(*
Nazwa:			VIS
Opis:			Zmienne wykorzystywane i zmieniane tylko z wizualizacji
Wersja:			v0.2
Data:			2024-02-06
Autor:			DP,MP
Urzadzenia:		
Konfiguracja:	
Info:
Zmiany:
- 20240205 [DP] Poprawki przed nowa wizką
*)

{attribute 'qualified_only'}

VAR_GLOBAL	
	
(********DANE MASZYNY***********)
sType: STRING[255];
sSerialNumber: STRING[255];
rProgramVersion: REAL;
rLastTimeChanges: REAL;
(*******************************)	

    (* OPISY ZMIENNYCH TYPU INT DO POŚWWIETLANIA STANÓW STACJI
	E_PackMLState : 
					eUndefined				:=  0, //----Nieużywany
					eClearing 				:=  1, //----Nieużywany
					eStopped 				:=  2, //Błąd
					eStarting 				:=  3, //Uruchamianie
					eIdle 					:=  4, //Postój
					eSuspended 				:=  5, //---Nieużywany
					eExecute 				:=  6, //Praca
					eStopping	 			:=  7, //Zatrzymywanie
					eAborting 				:=  8, //Zatrzymywanie awaryjne
					eAborted 				:=  9, //Zatrzymano awaryjnie
					eHolding 				:= 10, //---Nieużywany
					eHeld 					:= 11, //---Nieużywany
					eUnholding 				:= 12, //---Nieużywany
					eSuspending 			:= 13, //---Nieużywany
					eUnsuspending 			:= 14, //---Nieużywany
					eResetting 				:= 15, //Resetowanie błędu, bazowanie
					eCompleting 			:= 16, //---Nieużywany
					eComplete	 			:= 17  //---Nieużywany
	
	E_Station :
					eDisabled 				:= 0, // Stan nieaktywnosci (Stacja wyłączona)             
					eAborted 				:= 1, // Stan bezpiecznego zatrzymania (po Abortingu) 
					eAborting 				:= 2, // Stan bezpiecznego zatrzymywania (po EStopie)
					eError 					:= 3, // Stan błędu 		
					eResetting 				:= 4, // Stan resetowania bledu (po Errorze)		                
					eManualMovement 		:= 5, // Stan ruchów manualnych         
					eHoming 				:= 6, // Stan bazowania 
					eHomingDone 			:= 7, // Stan wykonania bazowania 
					ePreparingToReady 		:= 8, // Stan przygotowywania do gotowosci (zawsze przed Ready)           
					ePreparingToDisable 	:= 9, // Stan przygotowywania do nieaktywnosci (po wyłączeniu Enable)                               
					eReady					:= 10,// Stan gotowosci 
					eStopping 				:= 11,// Stan zatrzymywania 
					eStarting 				:= 12,// Stan uruchamiania (po Ready)
					eRunning 				:= 13 // Stan wykonywania cyklu (po Startingu), w tym stanie osobny 
					
					
	Legenda dla wizki :
	[H] - Hidden, prawdopodobnie nie potrzebne
	[I] - Info, informacja,
	[L] - Later, do zrobienia później, być może do przerobienia
	Uprawienia:
	brak opisu - operator
	[m] - Meechanik i powyżej
	[t] - Technolog i powyżej
	[s] - Serwis i powyżek
	[a] - Admin			
	*)
	(*****Zmienne ogólne****)
	
	(* Wykresy dozowania*)
	aPoints												: ARRAY [0..11,0..599] OF ST_Point;	// Sam wykres wybrando doziwniki + jego simulacji
	udiDossagerNum										: UDINT	:=	0;						// Wybrany dozownik 0 - pierwszy, 3 - czwarty
	bDrawChart											: BOOL;								// Cykl simulacji
	nDrawLenght										:INT;
	nTimeMarkerDSPh1                                :INT;
	nTimeMarkerDSPh2                                :INT;
	nTimeMarkerDSPh3                                :INT;
	nTimeMarkerDSPh4								:INT;
	nTimeMarkerDSPh5								:INT;
	aHorizontalChart								: ARRAY[0..4] OF ARRAY [0..0] OF INT;
	lrTorqMin										:LREAL;
	lrTorqMax										:LREAL;
	aWeightPoints									: ARRAY [0..7,0..9999] OF ST_Point_1;
	
	
	
	
	
	
	
	
	//Zmienne przejść do różnych stanów	
	iMachineState										:UINT;						// Stan maszyny
	sMachineState										:STRING; 					// Stan maszyny
	wsMachineState										:WSTRING; 					// Stan maszyny

	//Okno przezbrajania po wyborze receptury
	bMachinePartsChangeOver								:BOOL;						// Włączone przezbrajanie (ustawić z wizki)
	iMachinePartsChangeOver								:INT;						// Stan przezbrajania (0-ruch,1-pozycja gorna,-1-pozycja dolna) 
	bBottleSorterDisable								:BOOL:=FALSE;				// Wyłączenie sortera butelek
	bCapSorterDisable									:BOOL:=FALSE;				// Wyłączenie sortera nasadek
	
	//Ekran z komunikatami
	bDialogBoxOn										:BOOL;		 				// Wyświetl okno komunikatów
	bDialogBoxText										:STRING[255];				// Treść na oknie komunikatów 
	bDialogBoxText2										:STRING[255];				// Treść na oknie komunikatów (nie tłumaczone, zmienne)
	sDialogBoxPicture									:STRING[255];				// Nazwa obrazka który ma sie wyświetlać, '' - brak obrazu, 1,2,ok,info,uwaga 
																					// (odnosi się do pliku pictures.txt gdzie są podaje lokalizacje obrazków)
																					(*	[{"ImagePath":"c:\\img\\img1.png","ImageID":"1"}, 
																						{"ImagePath":"c:\\img\\img2.png","ImageID":"2"},
																						{"ImagePath":"c:\\img\\ok.png","ImageID":"ok"},
																						{"ImagePath":"c:\\img\\info.png","ImageID":"info"},
																						{"ImagePath":"c:\\img\\uwaga.png","ImageID":"uwaga"}] *)
	bDialogBoxAck										:BOOL;						// Przycisk OK
	bDialogBoxCancelAck									:BOOL;						// Przycisk ANULUJ
	nDialogBoxType										:UINT;						// Rodzaj okna, 0-nic, 1-tylko przycisk OK, 2 - tylko przycisk Anuluj, 3 - Przycisk OK i Anuluj
	bDialogBoxAckNeeded									:BOOL;						// [H] Potrzebne potwierdzenie					

	wsDialogBoxText										:WSTRING;				// Treść na oknie komunikatów 
	wsDialogBoxText2									:WSTRING;				// Treść na oknie komunikatów (nie tłumaczone, zmienne)
	
	//Wyświetlanie informacji na ekranie głównym
	//Przyczyny odrzuceń (wyświetlić na ekranie głównym bez dodatkowego odpisu)
	sBadPackageReason1									:STRING;					// Powód odrzutu butelek 		//sBadPackageReason1 sBadPackageReason1
	sBadPackageReason2									:STRING;					//								//sBadPackageReason2 sBadPackageReason2
	sBadPackageReason3									:STRING;					//								//sBadPackageReason3 sBadPackageReason3	
	iBadPackageReasonCount1								:INT;						// Ilość odrzuconych opakowań
	iBadPackageReasonCount2								:INT;						//
	iBadPackageReasonCount3								:INT;						//
	wsBadPackageReason1									:WSTRING;					// Powód odrzutu butelek 		//sBadPackageReason1 sBadPackageReason1
	wsBadPackageReason2									:WSTRING;					//								//sBadPackageReason2 sBadPackageReason2
	wsBadPackageReason3									:WSTRING;					//								//sBadPackageReason3 sBadPackageReason3	
	AStBadPackageReason									:ARRAY[0..63] OF S_Information;	// ID informacji do powodów odrzuceń
	bBadPackageReasonReset								:BOOL;						// Czyszczenie tablicy odrzuceń
	
	iNumbersOfFormsBetweenWeightAndScrewers				:INT;						// Ilość formatek pomiędzy wagą a zakręcarkami: zmienna
	
	sSlowestStation1									:STRING;					//	Najwolniejsza stacja nr 1	//sSlowestStation1 iSlowestStationCount1
	sSlowestStation2									:STRING;					//	Najwolniejsza stacja nr 2	//sSlowestStation2 iSlowestStationCount2
	sSlowestStation3									:STRING;					//	Najwolniejsza stacja nr 3	//itd.
	sSlowestStation4									:STRING;					//	Najwolniejsza stacja nr 4
	sSlowestStation5									:STRING;					//	Najwolniejsza stacja nr 5	
	iSlowestStationCount1								:INT;					  	//	Czas cyklu dla najwolniejszej stacji nr 1
	iSlowestStationCount2								:INT;					  	//	Czas cyklu dla najwolniejszej stacji nr 2
	iSlowestStationCount3								:INT;					  	//	Czas cyklu dla najwolniejszej stacji nr 3
	iSlowestStationCount4								:INT;					  	//	Czas cyklu dla najwolniejszej stacji nr 4
	iSlowestStationCount5								:INT;					  	//	Czas cyklu dla najwolniejszej stacji nr 5
	wsSlowestStation1									:WSTRING;					//	Najwolniejsza stacja nr 1	//sSlowestStation1 iSlowestStationCount1
	wsSlowestStation2									:WSTRING;					//	Najwolniejsza stacja nr 2	//sSlowestStation2 iSlowestStationCount2	
	wsSlowestStation3									:WSTRING;					//	Najwolniejsza stacja nr 3	//itd.	
	wsSlowestStation4									:WSTRING;					//	Najwolniejsza stacja nr 4	
	wsSlowestStation5									:WSTRING;					//	Najwolniejsza stacja nr 5	
	
	//Przyciski główne na HMI (wysuwany pasek lub na ekranie głównym)
	bDoorsUnlock										:BOOL;						// Otwórz drzwi 	
	bCycleReset											:BOOL;						// Reset cyklu 
	bCounterReset										:BOOL;						// Reset Liczników
	bConfectionEnding									:BOOL; 						// Zakończenie konfekcji
	bWeighingForm										:BOOL;						// [m] Przeważanie formatek
	bCapSorterEmptyingMode								:BOOL;						// Opróżnianie sortera nakrętek
	bBottleSorterEmptyingMode							:BOOL;						// Opróżnianie sortera butelek
	bBottleDeleteUnderDispencers						:BOOL;						// Usuń butelki pod dozownikami
	bSingleRealeseIfNoCapFromScrewers					:BOOL:=FALSE;						// Wypuszczanie pojedyńczo z zakręcarek jeżeli nie ma nasadki
	
	//Zmienne wystawiane z HMI
	bServiceMode										:BOOL; 						// Tryb serwisowy 
	bSimulation											:BOOL;						// [s] Przycisk trybu symulacyjnego
	bCheckStart 										:BOOL;						// Próba uruchomienia (PLC ustawia na 1, HMI na 0)
	bAllowStart 										:BOOL;						// Uruchomienie maszyny możliwe (HMI ustawia na 1 po bCheckStart i ktoś jest zalogowany, PLC ustawia na 0)
	iHMICommunication									:INT;						// [I] Licznik komunikacji, gdy się nie zmienia przez jakiś czas, wizka może wystawiać błąd
	bRecipeCalculate									:BOOL;						// Oblicz parametry receptury

	//[s] Zmienne tylko dla serwisu
	bWritePersistent									:BOOL; 						// [H] Zmienna zapisujaca wartosci zmiennych persistent
	bCycleStart											:BOOL;	(**)				// [H] Zdalny start/stop maszyny
	
	//Liczniki 
	uiCounterMachineEfficiency							:UINT; 						// Wydajność chwilowa maszyny[szt./h]
	uiCounterInstantEfficiency							:UINT; 						// Wydajność chwilowa prawidłowych butelek [szt./h]
	uiCounterAverageEfficiency							:UINT;						// Średnia wydajność [szt./h]
	udiCounterShiftBottles								:UDINT;						// Zmianowa ilość butelek [szt.]					
	uiCounterGoodBottles								:UINT;						// Prawidłowo napełnione opakowania [szt.]
	uiCounterBadBottles									:UINT;						// Odrzucone opakowania [szt]
	//Liczniki OEE
	udiCounterExecuteTime								:UINT;						// Cza pracy [min]
	udiCounterReadyTime									:UINT;						// Cza postoju [min]
	udiCounterErrorTime									:UINT;						// Cza błędu [min]
	
	//Lampki w trybie serwisowym pomocne do ustawiania stacji
	bCapPuttedCheckSensor								:BOOL;						// Czujnik nasadki przed zakręcarką
	bCapCorrectCheckCapOnSensor							:BOOL;						// Czujnik nasadki za zakręcarką
	bCapCorrectCheckCapNotScrewedSensor					:BOOL;						// Czujnik źle zakręconej nasadki

	(*Wykresy, statystyki, informacje*) 
	//Pomiary wag i dozowań do wyświetlenia na ekranie głównym
	lrDispencer1DoseVolumeCV							:LREAL;						// Doza 1 [ml]
	lrDispencer2DoseVolumeCV							:LREAL;						// Doza 2 [ml]
	lrDispencer3DoseVolumeCV							:LREAL;						// Doza 3 [ml]	
	lrDispencer4DoseVolumeCV							:LREAL;						// Doza 4 [ml]	
	lrDispencer1WeightMeasured							:LREAL;						// Waga z dozownika 1 [g]	
	lrDispencer2WeightMeasured							:LREAL;						// Waga z dozownika 2 [g]		
	lrDispencer3WeightMeasured							:LREAL;						// Waga z dozownika 3 [g]	
	lrDispencer4WeightMeasured							:LREAL;						// Waga z dozownika 4 [g]	
	bDispencer1WeightMeasured							:BOOL;						// [H] Waga zmierzona z dozownika nr 1	
	bDispencer2WeightMeasured							:BOOL;						// [H] Waga zmierzona z dozownika nr 2
	bDispencer3WeightMeasured							:BOOL;						// [H] Waga zmierzona z dozownika nr 3
	bDispencer4WeightMeasured							:BOOL;						// [H] Waga zmierzona z dozownika nr 4
		
	AsChartDose1										:ARRAY [0..500] OF STRING;	// [L] Wykres ostatniego dozowania 1 "Czas;PozycjaTłoka;PozycjaPodnośnika;ZawórSsący;ZaworDozujacy;Tacka" 
	AsChartDose2										:ARRAY [0..500] OF STRING;	// [L] Wykres ostatniego dozowania 2 "Czas;PozycjaTłoka;PozycjaPodnośnika;ZawórSsący;ZaworDozujacy;Tacka" 									
	AsChartDose3										:ARRAY [0..500] OF STRING;	// [L] Wykres ostatniego dozowania 3 "Czas;PozycjaTłoka;PozycjaPodnośnika;ZawórSsący;ZaworDozujacy;Tacka" 									
	AsChartDose4										:ARRAY [0..500] OF STRING;	// [L] Wykres ostatniego dozowania 4 "Czas;PozycjaTłoka;PozycjaPodnośnika;ZawórSsący;ZaworDozujacy;Tacka" 			
	AStAsChartDose1										:ARRAY [0..100] OF ARRAY [0..5,0..500] OF INT; // [L] Wykres ostatniego dozowania 1 "Czas;PozycjaTłoka;PozycjaPodnośnika;ZawórSsący;ZaworDozujacy;Tacka"
	AStAsChartDose2										:ARRAY [0..100] OF ARRAY [0..5,0..500] OF INT; // [L] Wykres ostatniego dozowania 1 "Czas;PozycjaTłoka;PozycjaPodnośnika;ZawórSsący;ZaworDozujacy;Tacka"
	AStAsChartDose3										:ARRAY [0..100] OF ARRAY [0..5,0..500] OF INT; // [L] Wykres ostatniego dozowania 1 "Czas;PozycjaTłoka;PozycjaPodnośnika;ZawórSsący;ZaworDozujacy;Tacka"
	AStAsChartDose4										:ARRAY [0..100] OF ARRAY [0..5,0..500] OF INT; // [L] Wykres ostatniego dozowania 1 "Czas;PozycjaTłoka;PozycjaPodnośnika;ZawórSsący;ZaworDozujacy;Tacka"
	
	
	AsChartGripperScrewer1								:ARRAY [0..500] OF STRING;	// [L] Wykres ostatniego zakręcania 1 "Czas;Wysokość;Obrót;Moment;SiłownikChwytania;;" 
	AsChartGripperScrewer2								:ARRAY [0..500] OF STRING;	// [L] Wykres ostatniego zakręcania 2 "Czas;Wysokość;Obrót;Moment;SiłownikChwytania;;" 
	AStChartGripperScrewer1								:ARRAY [0..100] OF ARRAY [0..5,0..500] OF INT;	// [L] Wykres ostatniego zakręcania 1 "Wysokość;Obrót;Prędkość;SiłownikChwytania;Czas;Pusty;;" 	
	AStChartGripperScrewer2								:ARRAY [0..100] OF ARRAY [0..5,0..500] OF INT;	// [L] Wykres ostatniego zakręcania 2 "Wysokość;Obrót;Prędkość;SiłownikChwytania;Czas;Pusty;;" 
	
	//[L] Przepisanie stanów wyjść ze sterownika na zmienne do HMI													
	//Pomiary przebiegu dozowania dozownika 1
	bHMIDispencer1SuckingValveActuator					:BOOL;						// Stan zaworu ssania dozownika nr 1
	bHMIDispencer1DosingValveActuator					:BOOL;						// Stan dozowania dozownika nr 1
	bHMIDispencer1DropCatcherValveActuator				:BOOL;						// Stan tacki dozownika nr 1
	//Pomiary przebiegu dozowania dozownika 2
	bHMIDispencer2SuckingValveActuator					:BOOL;						// Stan zaworu ssania dozownika nr 2
	bHMIDispencer2DosingValveActuator					:BOOL;						// Stan dozowania dozownika nr 2
	bHMIDispencer2DropCatcherValveActuator				:BOOL;						// Stan tacki dozownika nr 2
	//Pomiary przebiegu dozowania dozownika 3
	bHMIDispencer3SuckingValveActuator					:BOOL;						// Stan zaworu ssania dozownika nr 3
	bHMIDispencer3DosingValveActuator					:BOOL;						// Stan dozowania dozownika nr 3
	bHMIDispencer3DropCatcherValveActuator				:BOOL;						// Stan tacki dozownika nr 3
	//Pomiary przebiegu dozowania dozownika 4
	bHMIDispencer4SuckingValveActuator					:BOOL;						// Stan zaworu ssania dozownika nr 4
	bHMIDispencer4DosingValveActuator					:BOOL;						// Stan dozowania dozownika nr 4
	bHMIDispencer4DropCatcherValveActuator				:BOOL;						// Stan tacki dozownika nr 4
	//Prędkość podnośnika
	iHMIDispencersLifterMaxSpeed						:INT;						// Prędkość maksymalna podnośników dozowników (do ustawiania wykresów dozowników)

	//Tablica rejestrów z opisami
	AbFormPresent										:ARRAY [1..100] OF BOOL;	// Widoczność formatki formatki (np. .[2]=TRUE to formatka jest widoczna na 2 miejscu
	AsFormDescription									:ARRAY [1..100] OF STRING;	// Opis formatki (jedna literka, np. B,P,C) (.[2] to opis formatki na 2 miejscu)	
	                                        	
	(*****P00_Alarms***)    	                   									// Wyświetla tylko jeden błąd na raz, zatrzymuje maszynę    		                            	
	bErrorOccure										:BOOL:=FALSE;				// Błąd
	sStationInError										:STRING:='';				// Nazwa stacji
	udiStationInError									:UDINT:=0;					// ID Nazwa stacji która jest w stanie błędu 	//sStationName.xlsx
	udiStationErrorCode									:UDINT:=0;					// ID Kod błędu stacji							//sErrorString.xlsx
	sStationErrorDescription							:STRING(200):='';			// Opis błędu stacji - tłumaczony
	sStationErrorDescription2							:STRING(200):='';			// Opis błędu stacji - nie tłumaczony                    	
	bResetErrorVisuCmd									:BOOL:=FALSE;				// Reset błędu
	
	wsStationInError									:WSTRING:="";				// Nazwa stacji
	wsStationErrorDescription							:WSTRING(200):="";			// Opis 
	wsStationErrorDescription2							:WSTRING(200):="";			// Opis błędu (nie tłumaczony, zmienny)                      	

	fbAlarms 											:FB_Events;					// EventLogger

	//Warningi											// Wyświetlanie warningów, nie zatrzymuje maszyny	
	bWarningAcknowledgeAll								:BOOL;					 	// Przycisk potwierdzenia wszystkie ostrzeżenia
	bWarningNew											:BOOL;					 	// Pojawiło się nowe ostrzezenie 1s
	uliWarningOccure 									:ULINT;					 	// Wystąpienie ostrzezenia (każdy bit to inne ostrzeżenie [0..63])
	uliWarningAcknowledge 								:ULINT;						// Potwierdzenie ostrzezenia (każdy bit to inne ostrzeżenie [0..63])
	AsWarningDescription								:ARRAY [0..63] OF STRING;	// Opis ostrzeżenia (tablica na stałe wypisana)
															// VIS.AsWarningDescription[0]:='Niski pozom zbiornika nr 1';
															// VIS.AsWarningDescription[1]:='Niski pozom zbiornika nr 2';
															// VIS.AsWarningDescription[2]:='Zapełniony transproter odrzuconych opakowań';	
															// VIS.AsWarningDescription[3]:='			';
															// VIS.AsWarningDescription[4]:='Brak stabilizacji wagi przy pomiarach';
															// VIS.AsWarningDescription[5]:='Smarowanie robota';
															// VIS.AsWarningDescription[6]:='Brak odczytu RFID przed dozownikami';
															// VIS.AsWarningDescription[7]:='Brak odczytu RFID przed wagą';
															// VIS.AsWarningDescription[8]:='Brak odczytu RFID przed zakręcarką';
															// VIS.AsWarningDescription[9]:='Brak odczytu RFID pod robotem';

															// VIS.AsWarningDescription[10]:='Nieskalibrowany czujnik chwytaka szyjek pod dozownikami';
															// VIS.AsWarningDescription[11]:='Chwytak dozownika 1 - butelka nieprawidłowo chwycona';																					
															// VIS.AsWarningDescription[12]:='Chwytak dozownika 2 - butelka nieprawidłowo chwycona';																							
															// VIS.AsWarningDescription[13]:='Chwytak dozownika 3 - butelka nieprawidłowo chwycona';																							
															// VIS.AsWarningDescription[14]:='Chwytak dozownika 4 - butelka nieprawidłowo chwycona';	
															
															// VIS.AsWarningDescription[15]:='Zakręcarka 1 - przekroczenie czasu zakręcania - zmień ust.';		
															// VIS.AsWarningDescription[16]:='Zakręcarka 1 - przekroczenie czasu szukania gwintu - zmień ust.';
															// VIS.AsWarningDescription[17]:='Zakręcarka 1 - przekroczenie poślizgu - zmień ust.';
															// VIS.AsWarningDescription[18]:='Zakręcarka 1 - zbyt niska pozycja przy zakrecaniu - zmień ust.';
															// VIS.AsWarningDescription[19]:='Zakręcarka 2 - przekroczenie czasu zakręcania - zmień ust.';		
															// VIS.AsWarningDescription[20]:='Zakręcarka 2 - przekroczenie czasu szukania gwintu - zmień ust.';
															// VIS.AsWarningDescription[21]:='Zakręcarka 2 - przekroczenie poślizgu - zmień ust.';
															// VIS.AsWarningDescription[22]:='Zakręcarka 2 - zbyt niska pozycja przy zakrecaniu - zmień ust.';
															
	AwsActiveWarningDescription								:ARRAY [0..63] OF WSTRING;	//  Aktywne ostrzeżenia
	iActiveWarning											:INT;	// Ilość aktywnych ostrzeżeń				
	AudiActiveWarningDescriptionID							:ARRAY [0..63] OF UDINT;	// ID warningów do tłumaczeń na wizualizacji
																
	//Informacje // Pojawiają się na ekranie głównym i same znikają, jeżeli [0] > '' to wyświetl i usuń jak jest ''
	bInformationNew											:BOOL;					 		// Pojawiła sie nowa informacja
	AsInformationDescription  								:ARRAY[0..63] OF STRING; 		// Opis informacji, tablica na stałe wypisana
	iActiveInformation										:INT;					 		// Ilość aktywnych informacji
	AStInformationDescription								:ARRAY[0..63] OF S_Information;	// ID informacji do tłumaczeń na wizualizacji Struktura


																			
	(****P00_OEE*****) //Generowanie informacji do stworzenia OEE na wizualizacji
	// [L] Symbole według DescriptionStations.txt
	AsOEECycleTimes										:ARRAY [1..64] OF STRING;	// [L] Tabela czasów cykli 		[symbol_stacji;czas_w_ms] 	
	// Symbole według DecriptionRejectReason.txt
	// [L] Po ustawieniu powodu, dodawany jest ID
	sOEERejectionReason									:STRING;					// [L] Powód odrzuceń			[symbol_odrzucenia]

	sOEEText1											:STRING;					// Tekst 1			[PRACA:2h30MIN]
	sOEEText2											:STRING;					// Tekst 2			[POSTÓJ:1h30MIN]
	sOEEText3											:STRING;					// Tekst 1			[BŁĄD:2h30MIN]
	bOEEGenRaport										:BOOL;						//
	iOEEPackMLSuspendedReason							:INT;																																																																                                                        
	(**P01_BottleSorter***)
	// Sorter butelek
	bBottleSorterHold									:BOOL;
	// Zmienne czytane z innegro sterownika
	
	(***P01_BottleSorter***)
	// Podajnik butelek 
	iBottleFeederState									:INT;						// Stan
	sBottleFeederState									:STRING;					// Stan
	bBottleFeederRun									:BOOL;						// Cykl
	bBottleFeederHoming									:BOOL;						// Bazowanie 
	bBottleFeederIgnoreError							:BOOL;						// Ignoruj błędy
	bBottleFeederManualArmDown							:BOOL;						// Dół
	bBottleFeederManualArmLeft							:BOOL;						// Lewo
	bBottleFeederManualGate1							:BOOL;						// Szlaban 1 - lewy
	bBottleFeederManualGate2							:BOOL;						// Szlaban 2 - prawy
	bBottleFeederManualGripper							:BOOL;						// Chwytak
	bBottleFeederManualFormPositioning					:BOOL;						// Pozycjonowanie formatki
	bBottleFeederManualFormGate							:BOOL;						// Szlaban formatki		

	// Podajnik butelek - stół							
	iBottleFeederTurnTableState							:INT; 					 	// Stan
	sBottleFeederTurnTableState							:STRING; 					// Stan
	nBottleFeederTurnTableVelocityCV					:UDINT;						// Aktualna prędkość
	bBottleFeederTurnTableManualCmdStart				:BOOL; 					 	// Start 

	(***P01_PucksInserter***)
	// Podajnik opakowań
	iPucksInserterState									:INT;						// Stan
	sPucksInserterState									:STRING;					// Stan
	bPucksInserterRun									:BOOL;						// Cykl
	bPucksInserterHoming								:BOOL;						// Bazowanie 
	bPucksInserterHeightSet								:BOOL;						// Ustaw
	bPucksInserterIgnoreError							:BOOL;						// Ignoruj błędy
	bPucksInserterManualHammer							:BOOL;						// Wbijak	
	bPucksInserterManualTray							:BOOL;						// Tacka
	bPucksInserterManualGate1							:BOOL;						// Szlaban 1 - lewy
	bPucksInserterManualGate2							:BOOL;						// Szlaban 2 - prawy
	bPucksInserterManualFormGate						:BOOL;						// Szlaban formatki		
	bPucksInserterManualFormPositioning					:BOOL;						// Pozycjonowanie formatki	
	bPucksInserterManualWheelLeft						:BOOL;						// Karuzela - przód	
	bPucksInserterManualWheelRight						:BOOL;						// Karuzela - tył
	lrPucksInserterWheelPositionCV						:LREAl;						// Aktualna pozycja karuzeli


	//Transporter
	nPucksInserterConveyorVelocityCV					:UDINT;						// Aktualna prędkość
	bPucksInserterConveyorManualCmdStart				:BOOL; 					 	// Start 			
			
	// Wbijak na podnośniku
	lrPucksInserterHammerHeightCV						:LREAL;  					// Aktualna pozycja
    bPucksInserterManualHammerUp						:BOOL;  					// Do góry
    bPucksInserterManualHammerDown						:BOOL;  					// Na dół

	// Podajnik opakowań - stół							
	iPucksInserterTurnTableState						:INT; 					 	// Stan
	sPucksInserterTurnTableState						:STRING; 					// Stan
	nPucksInserterTurnTableVelocityCV					:UDINT;						// Aktualna prędkość
	bPucksInserterTurnTableManualCmdStart				:BOOL; 					 	// Start 
	
	
	//Stół popychający butelki Vasyl 27.05
	bPucksInserterPushTable_m1_ManualCmdStart				:BOOL; 					 	// Start silnik stołu pchającego - nr1
	bPucksInserterPushTable_m2_ManualCmdStart				:BOOL; 					 	// Start silnik stołu pchającego - nr2 
	bPucksInserterPushTable_m3_ManualCmdStart				:BOOL; 					 	// Start silnik stołu pchającego - nr3
	bPucksInserterPushTable_g1_ManualActuator				:BOOL;						// do usuniecia Siłownik stołu pchającego - nr1
	bPucksInserterPushTable_g2_ManualActuator				:BOOL;						// do usuniecia Siłownik stołu pchającego - nr2
	sPucksInserterPushTableState							:STRING;
	iPucksInserterPushTableState							:INT;
	sPucksInserterPushTableRollerState						:STRING;
	iPucksInserterPushTableRollerState						:INT;
	uiPucksInserterPushTable_m1_Velocity					:INT;
	uiPucksInserterPushTable_m2_Velocity					:INT;
	uiPucksInserterPushTable_m3_Velocity					:INT;
	
	(*****P01_Gates********)   
	// Szlaban przed dozownikami	
	iGateBeforeDispencersState							:INT; 						// Stan
	sGateBeforeDispencersState							:STRING; 					// Stan 
	bGateBeforeDispencersRun							:BOOL;						// Cykl
	bGateBeforeDispencersManualActuator					:BOOL;						// Manual - Szlaban
	
	(********P01_TwoPhasesBarriers*****)
	// Szlaban między dozownikami
	iBarrierBetweenDispencerState						:INT;						// Stan
	sBarrierBetweenDispencerState						:INT;						// Stan
	bBarrierBetweenDispencerRun							:BOOL;						// Cykl
	bBarrierBetweenDispencerManualActuator				:BOOL;						// Szlaban
	// Szlaban między wagami	
	iBarrierBetweenWeightState							:INT;						// Stan
	sBarrierBetweenWeightState							:INT;						// Stan
	bBarrierBetweenWeightRun							:BOOL;						// Cykl
	bBarrierBetweenWeightManualActuator					:BOOL;						// Szlaban
	// Szlaban przed wagą 1-4
	bGateBeforeWeight14Run								:BOOL;						// Cykl
	bGateBeforeWeight14ManualActuator					:BOOL;						// Szlaban
	// Szlaban przed wagą 5-6
	bGateBeforeWeight56Run								:BOOL;						// Cykl
	bGateBeforeWeight56ManualActuator					:BOOL;						// Szlaban
	// Szlaban przed podawaniem słoików	
	iBarrierLidFeederState								:INT;						// Stan
	sBarrierLidFeederState								:INT;						// Stan
	bBarrierLidFeederRun								:BOOL;						// Cykl
	bBarrierLidFeederManualActuator						:BOOL;						// Szlaban	
	// Szlaban przed podawaniem knotów	
	iBarrierWickFeederState								:INT;						// Stan
	sBarrierWickFeederState								:INT;						// Stan
	bBarrierWickFeederRun								:BOOL;						// Cykl
	bBarrierWickFeederManualActuator						:BOOL;						// Szlaban		
	//Szlaban pod robotem       	
	iGateRobotState										:INT; 						// Stan
	sGateRobotState										:STRING; 					// Stan
	bGateRobotEntranceRun								:BOOL;						// Cykl
	bGateRobotManualActuator							:BOOL;						// Szlaban
	
	(*[H]*P02_BottlePusher********)   
	// Wbijak butelek	
	iBottlePusherState									:INT; 						// [H] Stan
	sBottlePusherState									:STRING; 					// [H] Stan 
	bBottlePusherRun									:BOOL;						// [H] Cykl
	bBottlePusherManualActuator							:BOOL;						// [H] Manual - Szlaban	
	
	(*******P02_Dispencers******)
	// Przeciąganie formatek lewe
	iFormsDragingLeftState								:INT;						// Stan 
	sFormsDragingLeftState								:STRING;					// Stan  
	bFormsDragingLeftRun								:BOOL;						// Cykl
	bFormsDragingLeftHoming								:BOOL;						// Bazowanie 
	bFormsDragingLeftIgnoreError						:BOOL;						// Ignoruj błędy
	bFormsDragingLeftManualFork							:BOOL;						// Podnoszenie
	bFormsDragingLeftManualLeadBefore1					:BOOL;						// Prowadzenie 1
	bFormsDragingLeftManualLeadBefore2					:BOOL;						// Prowadzenie 2
	bFormsDragingLeftManualLeft							:BOOL;						// Przód
	bFormsDragingLeftManualRight						:BOOL;						// Tył
	lrFormsDragingLeftPositionCV						:LREAL;
	bFormsDispencersDragLeftMoveToEndPosition			:BOOL;
	// Przeciąganie formatek prawe	
	iFormsDragingRightState								:INT;						// Stan
	sFormsDragingRightState								:STRING;					// Stan 	
	bFormsDragingRightRun								:BOOL;						// Cykl
	bFormsDragingRightHoming							:BOOL;						// Bazowanie
	bFormsDragingRightIgnoreError						:BOOL;						// Ignoruj błędy
	bFormsDragingRightManualFork						:BOOL;						// Podnoszenie
	bFormsDragingRightManualLeadBefore1					:BOOL;						// Prowadzenie 1
	bFormsDragingRightManualLeadBefore2					:BOOL;						// Prowadzenie 2
	bFormsDragingRightManualLeft						:BOOL;						// Przód
	bFormsDragingRightManualRight						:BOOL;						// Tył
	lrFormsDragingRightPositionCV						:LREAL;
	bFormsDispencersDragRightMoveToEndPosition			:BOOL;
	//Dozowniki
 
	(**[L]**Synchronizacja dozowników**)
	//Przyśpieszenie obsługi dozowników
	//Synchronizacja potrzebna, po to aby wyświetlana aktualna pozycją się zgadzała
	//Po zaznaczeniu "synchronizacji jednego z dozowników" należy blokować przyciski aż zmienna "bDispencersSyncReady" będzie ustawiona (kilka sekund)
	//Na przykład: Jeżeli jest zaznaczone 1  i zostanie włączone "Dozuj" w PLC zostaje ustawiane "bDispencer1Dose"
	//Na przykład: Jeżeli jest zaznaczone SYNC 1 i 2 i zostanie włączone "Przeciągaj" w PLC zostaje ustawiane "bDispencer1PullingSlow","bDispencer2PullingSlow"
	//Na przykład: Jeżeli jest zaznaczone SYNC 3 i 4 i zostanie włączone "Dozuj" w PLC zostaje ustawiane "bDispencer3Dose","bDispencer4Dose"
	//itd. odpowiednio dla wszystkich przycisków trybu serwiswego
	bDispencer1Sync						: BOOL;			// Steruj 1 dozownikiem
	bDispencer2Sync						: BOOL;			// Steruj 2 dozownikiem
	bDispencer3Sync						: BOOL;			// Steruj 3 dozownikiem
	bDispencer4Sync						: BOOL;			// Steruj 4 dozownikiem
	bDispencer12Sync					: BOOL;			// Steruj 12 dozownikiem
	bDispencer34Sync					: BOOL;			// Steruj 34 dozownikiem
	bDispencer1234Sync					: BOOL;			// Steruj 1234 dozownikiem
	
	bDispencersSyncReady				: BOOL;			// Gotowość (odblokowane okienko sterowania)		

	// Zmienne ogólne okienka serwisowego, zależnie od zaznaczonych synchronizacji dozowników
    bDispencersDose                		: BOOL;   		// Dozuj
    bDispencersIgnoreErrors        		: BOOL;   		// Ignoruj błędy
    bDispencersHoming           		: BOOL;         // Bazowanie
    bDispencersManualDropCatcher 		: BOOL;         // Tacki
	bDispencersCleaning					: BOOL;			// Mycie
	lrDispencersManualOverride			: LREAL;		// [H] Prędkość
    bDispencersManualPistonBack     	: BOOL;   		// Tłok do góryw
    bDispencersManualPistonForward  	: BOOL;  		// Tłok w dół
    lrDispencersActPos             		: LREAL;  		// Aktualna pozycja tłoka
    bDispencersManualLifterUp       	: BOOL;   		// Podnośnik do góry
    bDispencersManualLifterDown   		: BOOL;   		// Podnośnik w dół
    lrDispencersLifterActPos      		: LREAL;  		// Aktualna pozycja 
    bDispencersPullingFast          	: BOOL;   		// Przeciąganie szybkie
    bDispencersPullingSlow         		: BOOL;   		// Przeciąganie wolne	
  	bDispencersPullingFastContinous		: BOOL;   		// Przeciąganie szybkie 30s
    bDispencersPullingSlowContinous		: BOOL;   		// Przeciąganie wolne 30s
    bDispencersManualSuckValve     		: BOOL;  	 	// Zawór ssący
    bDispencersManualDoseValve     		: BOOL;   		// Zawór tłoczący
	lrDispencersLifterSetPosStepMode	: LREAL;		// Skok ruchu [mm] (1.0-5.0)
	bDispencersLifterStepMode			: BOOL;			// Tryb krokowy
	//Ready position									
    bDispencersHeightSet          		: BOOL;   		// Ustaw
	(***Koniec synchronizacja dozowników**)	
	
	// [L] Mycie CIP 
	bDispencersCIP										: BOOL;						// [H] Włączone mycie CIP (stacje dozowników i chwytaków obniżają się)
	iDispencersCIP										: INT;						// [H] Zmienna pomocnicza od CIP (-1 pozycja dół, 0-Ruch, 1-pozycja górna)
	bDispencer12Cleaning								: BOOL;						// [H] Włączenie przeciągania dla dozownika 1 i 2 , wyłącza się po odciśnięciu przycisku
	bDispencer34Cleaning								: BOOL;						// [H] Włączenie przeciągania dla dozownika 3 i 4 , wyłącza się po odciśnięciu przycisku
	bDispencerManualDropCatcherSuck						: BOOL;						// Zasysanie z tacek

	//Podnośnik dozownika 1 2
    bDispencer12ManualLifterUp      					:BOOL;   					// Podnośnik 12 do góry
    bDispencer12ManualLifterDown  						:BOOL;   					// Podnośnik 12 w doł
	//Podnośnik dozownika 3 4
    bDispencer34ManualLifterUp      					:BOOL;   					// Podnośnik 34 do góry
    bDispencer34ManualLifterDown    					:BOOL;   					// Podnośnik 34 w dół

	lrDispencer12LifterActPos							:LREAL;						// Aktualna pozycja podnośnika dozownika 12
	lrDispencer12LifterSetPosStepMode					:LREAL;						// Krok przesuwania [mm] (1-5.0)
	bDispencer12LifterStepMode							:BOOL;						// Tryb krokowy
	
	lrDispencer34LifterActPos							:LREAL;						// Aktualna pozycja podnośnika dozownika 34
	lrDispencer34LifterSetPosStepMode					:LREAL;						// Krok przesuwania [mm] (1-5.0)
	bDispencer34LifterStepMode							:BOOL;						// Tryb krokowy

	
	bDispencer12LifterHeightSet							: BOOL;						// Ustaw podnośnik 12
	bDispencer34LifterHeightSet							: BOOL;						// Ustaw podnośnik 34
	
	//Dozownik 1                                        
	iDispencer1State									:INT; 						// Stan
	sDispencer1State									:STRING; 					// Stan
	bDispencer1IgnoreErrors								:BOOL; 						// Ignoruj błędy	
	bDispencer1Dose										:BOOL; 						// Dozuj 1
	lrDispencer1ActPos									:LREAL;						// Aktualna pozycja tłoka 1
	bDispencer1PullingFast								:BOOL;						// Przeciągnie szybkie 1
	bDispencer1PullingSlow								:BOOL;						// Przeciągnie wolne 1
	bDispencer1ManualPistonBack							:BOOL;						// Tłok 1 do góry
	bDispencer1ManualPistonForward						:BOOL;						// Tłok 1 w dół
	bDispencer1ManualSuckValve							:BOOL;						// Zawór ssący 1
	bDispencer1ManualDoseValve							:BOOL;						// Zawór dozujący 1

	//Dozownik 2                                        
	iDispencer2State									:INT; 						// Stan
	sDispencer2State									:STRING; 					// Stan
	bDispencer2IgnoreErrors								:BOOL; 						// Ignoruj błędy		
	bDispencer2Dose										:BOOL; 						// Dozuj 2
	lrDispencer2ActPos									:LREAL;						// Aktualna pozycja tłoka 2
	bDispencer2PullingFast								:BOOL;						// Przeciągnie szybkie 2
	bDispencer2PullingSlow								:BOOL;						// Przeciągnie wolne 2
	bDispencer2ManualPistonBack							:BOOL;						// Tłok 2 do góry
	bDispencer2ManualPistonForward						:BOOL;						// Tłok 2 w dół
	bDispencer2ManualSuckValve							:BOOL;						// Zawór ssący 2
	bDispencer2ManualDoseValve							:BOOL;						// Zawór dozujący 2

	//Dozownik 3                                        
	iDispencer3State									:INT; 						// Stan
	sDispencer3State									:STRING; 					// Stan
	bDispencer3IgnoreErrors								:BOOL; 						// Ignoruj błędy	
	bDispencer3Dose										:BOOL; 						// Dozuj 13
	lrDispencer3ActPos									:LREAL;						// Aktualna pozycja tłoka 3
	bDispencer3PullingFast								:BOOL;						// Przeciągnie szybkie 3
	bDispencer3PullingSlow								:BOOL;						// Przeciągnie wolne 3
	bDispencer3ManualPistonBack							:BOOL;						// Tłok 3 do góry
	bDispencer3ManualPistonForward						:BOOL;						// Tłok 3 w dół
	bDispencer3ManualSuckValve							:BOOL;						// Zawór ssący 3
	bDispencer3ManualDoseValve							:BOOL;						// Zawór dozujący 3
	                                                                                   
	//Dozownik 4                                        
	iDispencer4State									:INT; 						// Stan
	sDispencer4State									:STRING; 					// Stan
	bDispencer4IgnoreErrors								:BOOL; 						// Ignoruj błędy	
	bDispencer4Dose										:BOOL; 						// Dozuj 4
	lrDispencer4ActPos									:LREAL;						// Aktualna pozycja tłoka 4
	bDispencer4PullingFast								:BOOL;						// Przeciągnie szybkie 4
	bDispencer4PullingSlow								:BOOL;						// Przeciągnie wolne 4
	bDispencer4ManualPistonBack							:BOOL;						// Tłok 4 do góry
	bDispencer4ManualPistonForward						:BOOL;						// Tłok 4 w dół
	bDispencer4ManualSuckValve							:BOOL;						// Zawór ssący 4
	bDispencer4ManualDoseValve							:BOOL;						// Zawór dozujący 4
                                               
	//Podnośnik chwytaka                    	 
	lrDispencersCatchHeightCV							:LREAL;						// Aktualna wysokość chwytaka
    bDispencersCatchManualUp							:BOOL;  					// Do góry
    bDispencersCatchManualDown							:BOOL;  					// W dół
	bDispencersCatchHeightSet							:BOOL;						// Ustaw
	bDispencersCatchOpenCalibration						:BOOL;						// Kalibruj otwarcie
	bDispencersCatchCloseCalibration					:BOOL;						// Kalibruj zamknięcie
	
	//Podnośnik chwytaka i tacki 1                     	 
	iDispencersCatch1State								:INT;						// Stan
	sDispencersCatch1State								:STRING;					// Stan
	bDispencers1Catch									:BOOL;  					// Cykl
	bDispencersCatch1ManualActuator						:BOOL;  					// Chwytak
	
	//Podnośnik chwytaka i tacki 2                     	 
	iDispencersCatch2State								:INT;						// Stan
	sDispencersCatch2State								:STRING;					// Stan
	bDispencers2Catch									:BOOL;  					// Cykl
	bDispencersCatch2ManualActuator						:BOOL;  					// Chwytak
	
	//Podnośnik chwytaka i tacki 3                   	 
	bDispencers3Catch									:BOOL;  					// Stan
	iDispencersCatch3State								:INT;						// Stan
	sDispencersCatch3State								:STRING;					// Cykl
	bDispencersCatch3ManualActuator						:BOOL;  					// Chwytak

	//Podnośnik chwytaka i tacki 4                   	 
	iDispencersCatch4State								:INT;						// Stan
	sDispencersCatch4State								:STRING;					// Stan
	bDispencers4Catch									:BOOL;  					// Cykl
	bDispencersCatch4ManualActuator						:BOOL;  					// Chwytak

	//Zbiornik 1                                
	bTanksIgnoreError         					        :BOOL; 						// [H] Ignoruj błedy
    bTank1ManualMixer                 					:BOOL; 						// Mieszadło
    bTank1ManualHeater                					:BOOL; 						// Grzanie
    bTank1ManualSupplyPump            					:BOOL; 						// Pompa
    bTank1ManualPressure              					:BOOL; 						// Nadciśnienie
	lrTankHeatingTempCV									:LREAL;						// Temperatura zbiornika
	
	//Czujnik zbiornika 1
 	bTank1LevelSensorCalibrationLight					:BOOL;						// Kalibracja na pusto
	bTank1LevelSensorCalibrationDark					:BOOL;						// Kalibracja na pełno
	bHMITank1LevelSensorPumpOn							:BOOL;						// [I] Poziom (pompa załączona)
	iTank1LevelSensorValue								:INT; 						// Poziom [mm]
    bTank1LevelSensorHigh                               :BOOL;                      // [L] Zadany poziom ustawiony na 80%
    bTank1LevelSensorLow                                :BOOL;                      // [L] Zadany poziom ustawiony na 10%

	//Zbiornik 2  
    bTank2ManualMixer                 					:BOOL; 						// [H] Mieszadło
    bTank2ManualHeater                					:BOOL; 						// [H] Grzałka
    bTank2ManualSupplyPump            					:BOOL; 						// Pompa
    bTank2ManualPressure              					:BOOL; 						// [H] Nadciśnienie

	//Czujnik zbiornika 2
 	bTank2LevelSensorCalibrationLight					:BOOL;						// Kalibracja na pusto
	bTank2LevelSensorCalibrationDark					:BOOL;						// Kalibracja na pełno	
	bHMITank2LevelSensorPumpOn							:BOOL;						// [I] Poziom (pompa załączona)
	iTank2LevelSensorValue								:INT; 						// Poziom [mm]
     
	//Dodatkowe zbiorniki
	bHMITank3LevelSensorPumpOn							:BOOL;						// [I] Poziom (pompa załączona)
	iTank3LevelSensorValue								:INT; 						// Poziom [mm]
 	bHMITank4LevelSensorPumpOn							:BOOL;						// [I] Poziom (pompa załączona)
	iTank4LevelSensorValue								:INT; 						// Poziom [mm]
   
                                       	
	(*******P05_Weight*******)
	//Podnoszenie wag 
	iWeightLiftState									:INT;						// Stan 
	sWeightLiftState									:STRING;					// Stan 
	bWeightLiftRun										:BOOL;						// Cykl
	bWeightLiftHoming									:BOOL;						// Bazowanie
	//Waga 1 podnoszenie
	bWeight1ActuatorManualUp							: BOOL;						// Do góry
	bWeight1ActuatorManualDown							: BOOL;						// Na dół
	//Waga 2 podnoszenie
	bWeight2ActuatorManualUp							: BOOL;						// Do góry
	bWeight2ActuatorManualDown							: BOOL;						// Na dół
	//Waga 3 podnoszenie
	bWeight3ActuatorManualUp							: BOOL;						// Do góry
	bWeight3ActuatorManualDown							: BOOL;						// Na dół
	//Waga 4 podnoszenie	
	bWeight4ActuatorManualUp							: BOOL;						// Do góry
	bWeight4ActuatorManualDown							: BOOL;						// Na dół	
	//Waga 5 podnoszenie	
	bWeight5ActuatorManualUp							: BOOL;						// Do góry
	bWeight5ActuatorManualDown							: BOOL;						// Na dół	
	//Waga 6 podnoszenie	
	bWeight6ActuatorManualUp							: BOOL;						// Do góry
	bWeight6ActuatorManualDown							: BOOL;						// Na dół	
	
     //Waga 1                                                   
	iWeight1State										:INT;						// Stan
	sWeight1State										:STRING;					// Stan
	bWeight1DoWeighting									:BOOL;						// Ważenie
	bWeight1Tare										:BOOL;						// Taruj
	lrWeight1Measured									:LREAL;						// Waga [g]
	lrWeight1Mass										:LREAL;						// Waga masy [g] (na ekranie głównym)
	//Waga 2
	iWeight2State										:INT;						// Stan
	sWeight2State										:STRING;					// Stan
	bWeight2DoWeighting									:BOOL;						// Ważenie
	bWeight2Tare										:BOOL;						// Taruj
	lrWeight2Measured									:LREAL;						// Waga [g]
	lrWeight2Mass										:LREAL;						// Waga masy [g] (na ekranie głównym)
	//Waga 3
	iWeight3State										:INT;						// Stan
	sWeight3State										:STRING;					// Stan
	bWeight3DoWeighting									:BOOL;						// Ważenie
	bWeight3Tare										:BOOL;						// Taruj
	lrWeight3Measured									:LREAL;						// Waga [g]
	lrWeight3Mass										:LREAL;						// Waga masy [g] (na ekranie głównym)
	//Waga 4
	iWeight4State										:INT;						// Stan
	sWeight4State										:STRING;					// Stan
	bWeight4DoWeighting									:BOOL;						// Ważenie
	bWeight4Tare										:BOOL;						// Taruj
	lrWeight4Measured									:LREAL;						// Waga [g]
	lrWeight4Mass										:LREAL;						// Waga masy [g] (na ekranie głównym)
	//Waga 5	
	iWeight5State										:INT;						// Stan
	sWeight5State										:STRING;					// Stan
	bWeight5DoWeighting									:BOOL;						// Ważenie
	bWeight5Tare										:BOOL;						// Taruj
	lrWeight5Measured									:LREAL;						// Waga [g]
	lrWeight5Mass										:LREAL;						// Waga masy [g] (na ekranie głównym)
	//Waga 6
	iWeight6State										:INT;						// Stan
	sWeight6State										:STRING;					// Stan
	bWeight6DoWeighting									:BOOL;						// Ważenie
	bWeight6Tare										:BOOL;						// Taruj
	lrWeight6Measured									:LREAL;						// Waga [g]
	lrWeight6Mass										:LREAL;						// Waga masy [g] (na ekranie głównym)
	                                               
	(*****P05_WeightCorrection******)       
	//Korekcja wag            
	lrDispencer1CorrectionWeight						:LREAL;						// Korekta 1 [ml] (możliwosć edycji)
	lrDispencer2CorrectionWeight						:LREAL;						// Korekta 2 [ml] (możliwosć edycji)
	lrDispencer3CorrectionWeight						:LREAL;						// Korekta 3 [ml] (możliwosć edycji)
	lrDispencer4CorrectionWeight						:LREAL;						// Korekta 4 [ml] (możliwosć edycji)	
	bWeightCorrectionReset								:BOOL;						// Reset

	(*****P06_WickFeeder******)   	
	//Podajnik knotów
	iWickFeederState									: INT;         	// [E_Station] Stan pracy ogólny
	sWickFeederState									: STRING;       // [E_Station] Stan pracy ogólny
	bWickFeederHoming									: BOOL; 		// Wykonanie procedury bazowania podajnika knotów
	bWickFeederHeightSet								: BOOL; 		// Ustawianie wysokoci podnonika podajnika knotów
	lrWickFeederHeightCV								: LREAL; 		// Aktualna wysokoć 
	bWickFeederIgnoreErrors								: BOOL;     	// Ignorowanie błędów dozownika 1 i po wykonaniu pracy ustawienie że wszystko zostało zrobione

	bWickFeederSorterRun								: BOOL; 		// Sortuj
	bWickFeeder1PrepareRun								: BOOL; 		// Pre-Cykl1
	bWickFeeder1Run										: BOOL; 		// Cykl 1
	bWickFeeder2PrepareRun								: BOOL; 		// Pre-Cykl2
	bWickFeeder2Run										: BOOL; 		// Cykl 2

	bWickFeederManualHeightUp							: BOOL; 		// Do góry
	bWickFeederManualHeightDown							: BOOL; 		// Na dół
	bWickFeederManualSorterEngine						: BOOL;			// Sorter
	bWickFeederManualSorterAir							: BOOL;			// Wydmuch
	bWickFeederManualStopper							: BOOL;			// Stoper 
	bWickFeederManualStopper2							: BOOL;			// Stoper2 	
	bWickFeederManualSeparator1							: BOOL;			// Separator tor 1
	bWickFeederManualSeparator2							: BOOL;			// Separator tor 2
	bWickFeederManualSleve1SeparatorActIn				: BOOL;			// Separator tor 1 - rękaw
	bWickFeederManualSleve1SeparatorActOut				: BOOL;			// Separator tor 1 - butelka
	bWickFeederManualSleve2SeparatorActIn				: BOOL;			// Separator tor 2 - rękaw
	bWickFeederManualSleve2SeparatorActOut				: BOOL;			// Separator tor 2 - butelka
	bWickFeederManualHammer1							: BOOL;			//	Wbijak 1 
	bWickFeederManualHammer2							: BOOL;			//	Wbijak 2
	bWickFeederManualFormPositioning					: BOOL;			// Pozycjonowanie formatek

	//Podawanie knotów - przeciąganie	
	iWickFeederDragingStationState						: INT;
	sWickFeederDragingStationState						: STRING;						// Stan 
	bWickFeederDragingStationRun						: BOOL;							// Cykl
	bWickFeederDragingHoming							: BOOL;							// Bazowanie 
	bWickFeederDragingIgnoreError						: BOOL;							// Ignoruj błędy
	bWickFeederDragingManualFork						: BOOL;							// Podnoszenie
	bWickFeederDragingManualLeadBefore1					: BOOL;							// Prowadzenie 1
	bWickFeederDragingManualLeadBefore2					: BOOL;							// Prowadzenie 2
	bWickFeederDragingManualLeft						: BOOL;							// Przód
	bWickFeederDragingManualRight						: BOOL;							// Tył
	bFormsWickFeederDragMoveToEndPosition				: BOOL;                              	
	lrWickFeederDragingStationPositionCV				: LREAL; 

                                             
	(*****P06_LidFeeder******)   	
	//Podajnik platynek
	bLidFeederHoming									: BOOL; 						// Wykonanie procedury bazowania podajnika platynek
	bLidFeederHeightSet									: BOOL; 						// Ustawianie wysokoci podnonika podajnika platynek
	lrLidFeederHeightCV									: LREAL; 						// Aktualna wysokoć stacji podajnika platynek
	bLidFeederIgnoreErrors								: BOOL;     					// Ignorowanie błędów dozownika 1 i po wykonaniu pracy ustawienie że wszystko zostało zrobione
	bLidFeederManualHeightUp							: BOOL; 					 	// Ręczne podnoszenie stacji podajnika platynek
	bLidFeederManualHeightDown							: BOOL; 
	bLidFeederManualFormPositioning						: BOOL;							// Pozycjonowanie formatek pod podawaniem platynek.
	lrFeederDragingStationPositionCV					:LREAL; 

	//Podajnik platynek 1	
	iLidFeeder1State									: INT;         					// [E_Station] Stan pracy ogólny
	sLidFeeder1State									: STRING;         				// [E_Station] Stan pracy ogólny
	bLidFeeder1PrepareRun								: BOOL; 						// Rozkaz pobrania platynki
	bLidFeeder1Run										: BOOL; 						// Rozkaz odłożenia platynki
	lrLidFeeder1HeaterTempCV							: LREAL;						// Temperatura aktualna grzałki podajnika platynek
	bLidFeeder1ManualAct								: BOOL; 						// Ruch ręczny podajnika platynek
	bLidFeeder1ManualAct2								: BOOL; 						// Ruch ręczny siłownika drugiego podajnika platynek
	bLidFeeder1ManualSuckerAct							: BOOL; 						// Ręczne uruchomienie ssawki podajnika platynek
	bLidFeeder1ManualHeaterAct							: BOOL; 						// Ręczne uruchomienie siłownika grzałki podajnika platynek

	//Podajnik platynek 2
	iLidFeeder2State									: INT;         					// [E_Station] Stan pracy ogólny
	sLidFeeder2State									: STRING;         				// [E_Station] Stan pracy ogólny
	bLidFeeder2PrepareRun								: BOOL; 						// Rozkaz pobrania platynki
	bLidFeeder2Run										: BOOL; 						// Rozkaz odłożenia platynki
	lrLidFeeder2HeaterTempCV							: LREAL;						// Temperatura aktualna grzałki podajnika platynek
	bLidFeeder2ManualAct								: BOOL; 						// Ruch ręczny podajnika platynek
	bLidFeeder2ManualAct2								: BOOL; 						// Ruch ręczny siłownika drugiego podajnika platynek
	bLidFeeder2ManualSuckerAct							: BOOL; 						// Ręczne uruchomienie ssawki podajnika platynek
	bLidFeeder2ManualHeaterAct							: BOOL; 						// Ręczne uruchomienie siłownika grzałki podajnika platynek
		
	//Podawanie platynek przeciąganie	
	iLidFeederDragingStationState						: INT;
	sLidFeederDragingStationState						: STRING;					// Stan 
	bLidFeederDragingStationRun							: BOOL;						// Cykl
	bLidFeederDragingHoming								: BOOL;						// Bazowanie 
	bLidFeederDragingIgnoreError						: BOOL;						// Ignoruj błędy
	bLidFeederDragingManualFork							: BOOL;						// Podnoszenie
	bLidFeederDragingManualLeadBefore1					: BOOL;						// Prowadzenie 1
	bLidFeederDragingManualLeadBefore2					: BOOL;						// Prowadzenie 2
	bLidFeederDragingManualLeft							: BOOL;						// Przód
	bLidFeederDragingManualRight						: BOOL;						// Tył
	bFormsLidFeederDragMoveToEndPosition				: BOOL;                              		

	
	//Sprawdzanie platynki
    iLidPuttedCheckState            					: INT;    						// [E_Station] Stan pracy
    sLidPuttedCheckState            					: STRING; 						// Opis stanu pracy
	bLidPuttedCheckRun									: BOOL; 						// Sprawdź
    bLidPuttedCheckHoming           					: BOOL;   						// Bazowanie stacji sprawdzania nasadek
    bLidPuttedCheckHeightSet        					: BOOL;   						// Ustawianie wysokoci stacji sprawdzania nasadek
    bLidPuttedCheckIgnoreErrors     					: BOOL;   						// Ignorowanie błędów stacji sprawdzania nasadek i po wykonaniu pracy ustawienie że wszystko zostało zrobione
    lrLidPuttedCheckHeightCV        					: LREAL;  						// Aktualna wysokoć stacji sprawdzania nasadek
	lrLidPuttedCheckSetPosStepMode						: LREAL;						// Tryb manualny, Ruch podnośnika o zadaną wartość z VIS w trybie krokowym
	bLidPuttedCheckStepMode		 						: BOOL;							// Trzyb manualny, Sterowanie napędem w trybie krokowym.
    bLidPuttedCheckManualHeightUp   					: BOOL;							// Ręczne podnoszenie stacji sprawdzania nasadek
    bLidPuttedCheckManualHeightDown 					: BOOL;							// Reczne opuszczanie stacji sprawdzania nasadek
	bLidPuttedCheckOK									: BOOL;							// Plantyka OK
	AsLidPuttedCheckProgramDescription					: ARRAY [0..20] OF STRING;		// Opis programów kamer, 0 - Opis programu nr 1, 1 - Opis programu nr 2
	
	//Grzałka zasadnicza                                
    bLidSealerHoming									: BOOL;							// Bazowanie stacji zgrzewania zasadniczego
    bLidSealerIgnoreErrors								: BOOL;						    // Ignorowanie błędów Zgrzewarki i po wykonaniu pracy ustawienie że wszystko zostało zrobione
  	lrLidSealerHeightCV									: LREAL;						// Aktualna wysokoć stacji zgrzewania zasadniczego
 	bLidSealerHeightSet									: BOOL;							// Ustawianie wysokości zgrzewarki
    bLidSealerManualHeightUp							: BOOL; 					    // Ręczne podnoszenie stacji grzałki zasadniczej
    bLidSealerManualHeightDown							: BOOL;					    	// Reczne opuszczanie stacji grzałki zasadniczej

	//Grzałka zasadnicza 1                               
	iLidSealer1State									: INT;							// [E_Station] Stan pracy ogólny
	sLidSealer1State									: STRING;						// [E_Station] Stan pracy ogólny
	bLidSealer1Run										: BOOL;							// Rozkaz zgrzania platynki
  	lrLidSealer1HeaterTempCV							: LREAL;						// Temperatura aktualna grzałki zasadniczej
    bLidSealer1ManualAct								: BOOL;							// Ruch ręczny grzałki zasadniczej

	//Stoper
	bLidSealerStoperManualActuator						: BOOL;
	
	//Grzałka zasadnicza 2
	iLidSealer2State									: INT;							// [E_Station] Stan pracy ogólny
	sLidSealer2State									: STRING;						// [E_Station] Stan pracy ogólny
	bLidSealer2Run										: BOOL;							// Rozkaz zgrzania platynki
  	lrLidSealer2HeaterTempCV							: LREAL;						// Temperatura aktualna grzałki zasadniczej
    bLidSealer2ManualAct								: BOOL;							// Ruch ręczny grzałki zasadniczej
		
	//Zgrzanie platynek przeciąganie	
	iLidSealerDragingStationState						: INT;
	sLidSealerDragingStationState						: STRING;					// Stan  
	bLidSealerDragingStationRun							: BOOL;						// Cykl
	bLidSealerDragingHoming								: BOOL;						// Bazowanie
	bLidSealerDragingIgnoreError						: BOOL;						// Ignoruj błędy
	bLidSealerDragingManualFork							: BOOL;						// Podnoszenie
	bLidSealerDragingManualLeadBefore1					: BOOL;						// Prowadzenie 1
	bLidSealerDragingManualLeadBefore2					: BOOL;						// Prowadzenie 2
	bLidSealerDragingManualLeft							: BOOL;						// Przód
	bLidSealerDragingManualRight						: BOOL;						// Tył
	lrSealerDragingStationPositionCV					:LREAL;
	bFormsLidSealerDragMoveToEndPosition			:BOOL;
	
	(*****P08_CapFeeder********)
	// [H] Podajnik nakrętek
	iCapFeederState										:INT;						// [H] Stan
	sCapFeederState										:STRING;					// [H] Stan
    bCapFeederHoming									:BOOL;						// [H] Bazowanie
 	bCapFeederRun										:BOOL; 						// [H] Cykl
	bCapFeederIgnoreErrors								:BOOL;					 	// [H] Ignoruj błędy
	bCapFeederHeightSet									:BOOL;						// [H] Ustaw
	bCapFeederManualHeightUp							:BOOL;						// [H] Do góry
	bCapFeederManualHeightDown							:BOOL;						// [H] Na doł
	bCapFeederManualSorterEngine						:BOOL;						// [H] Silnik
	bCapFeederManualSorterAir							:BOOL;						// [H] Wydmuch
	lrCapFeederHeightCV									:LREAL;						// [H] Aktualna wyskokość 
	bCapFeederManualGate1								:BOOL;						// [H] Szlaban 1
	bCapFeederManualGate2								:BOOL;						// [H] Szlaban 2				                                			

	(*****P08_CapSorter********)	 
	bCapSorterHold										:BOOL; 
	// Przeciąganie formatek pod sorterem nakrętek
	iCapSorterDragState									:INT;						// Stan
	sCapSorterDragState									:STRING;					// Stan
	bCapSorterDragRun									:BOOL;						// Cykl
	bCapSorterDragHoming								:BOOL;						// Bazowanie 
	bCapSorterDragIgnoreError							:BOOL;						// Ignoruj błędy
	bCapSorterDragManualFork							:BOOL;						// Podnosnik
	bCapSorterDragManualLeadBefore1						:BOOL;						// Prowadzenie
	bCapSorterDragManualLeadAfter1						:BOOL;
	bCapSorterDragManualLeft							:BOOL;						// Do przodu
	bCapSorterDragManualRight							:BOOL;						// Do tyłu
	lrCapSorterDragPositionCV							:LREAL;
	bFormsCapSorterDragMoveToEndPosition			:BOOL;
	//Stoper
	bCapSorterStoperManualActuator						: BOOL;

	(*****P09_CapPuttedCheck********) 
	// Sprawdzanie nasadki               			
	iCapPuttedCheckState								:INT;         				// Stan
	sCapPuttedCheckState								:STRING;         			// Stan
    bCapPuttedCheckHoming								:BOOL;					   	// Bazowanie
    bCapPuttedCheckIgnoreErrors							:BOOL := FALSE;				  // Ignoruje błędy
   	lrCapPuttedCheckHeightCV							:LREAL;				 		// Aktualna wysokoć 
    bCapPuttedCheckManualHeightUp						:BOOL; 						// Do góry
    bCapPuttedCheckManualHeightDown						:BOOL;			 			// Na dół
	bCapPuttedCheckHeightSet							:BOOL;						// Ustaw

 	(*****P10_GripperScrewer********)
	//Przeciąganie formatek po zakręcarkami
	iBottleDragingStationState							:INT;						// Stan 
	sBottleDragingStationState							:STRING;					// Stan 
	bBottleDragingStationRun							:BOOL;						// Cykl
	bBottleDragingStationHoming							:BOOL;						// Bazowanie
	bBottleDragingStationIgnoreError					:BOOL;						// Ignoruj błędy
	bBottleDragingStationManualFork1					:BOOL;						// Podnoszenie
	bBottleDragingStationManualLead						:BOOL;						// Prowadzenie
	bBottleDragingStationManualLeft						:BOOL;						// Do przodu
	bBottleDragingStationManualRight					:BOOL;						// Do tyłu
	lrBottleDragingStationPositionCV					:LREAL;
	bFormsScrewersDragMoveToEndPosition				:BOOL;
	
	//Zakręcarki szczękowe 
    bGripperScrewerIgnoreErrors							:BOOL; 						// Ignoruj błędy
  	bGripperScrewerHoming								:BOOL;						// Bazowanie
	bGripperScrewerHeightSet							:BOOL;						// Ustaw
	lrGripperScrewerManualOverride						:LREAL:=100;  				// [H] Prędkość
	AsGripperScrewerTool								:ARRAY [0..10] OF STRING;	// Głowica (1-Opis_narzędzia_nr_1, 2-Opis_narzędzia_nr_2)

	//Zakręcarka 1
	iGripperScrewer1State								:INT;						// Stan
	sGripperScrewer1State								:STRING;					// Stan
	lrGripperScrewer1LiftActPos							:LREAL;	 	  				// Aktualna pozycja
  	bGripperScrewer1Run									:BOOL;						// Cykl
    bGripperScrewer1ManualRight							:BOOL;  					// Obrót w prawo
    bGripperScrewer1ManualLeft							:BOOL;   					// Obrót w lewo
    bGripperScrewer1ManualCatch							:BOOL;  					// Chwyć
  	bGripperScrewer1AdjustTorque						:BOOL;						// [H] Badanie momentu odkręcania
	lrGripperScrewer1AdjustingSetTorque					:LREAL := 1.0;				// [H] Zadany szukany moment otwierania [Nm]
	lrGripperScrewer1TorqueCV							:LREAL;  					// Moment dokręcenia [nM] (po zakręceniu)

	//Zakręcarka 2	
	iGripperScrewer2State								:INT;						// Stan
	sGripperScrewer2State								:STRING;					// Stan
	lrGripperScrewer2LiftActPos							:LREAL;	 	  				// Aktualna pozycja
	bGripperScrewer2Run									:BOOL;                      // Cykl
    bGripperScrewer2ManualRight							:BOOL;  					// Obrót w prawo
    bGripperScrewer2ManualLeft							:BOOL;   					// Obrót w lewo
    bGripperScrewer2ManualCatch							:BOOL;  					// Chwyć
	lrGripperScrewer2TorqueCV							:LREAL;  					// Moment dokręcenia [nM] (po zakręceniu)

	bGripperScrewer1SetPositionOffset					:BOOL;						// Ustaw offset 1
	bGripperScrewer2SetPositionOffset					:BOOL;						// Ustaw offset 2
	
	//Podnośnik zakręcarek
	bGripperScrewerLiftManualHeightUp					:BOOL;  					// Do góry
    bGripperScrewerLiftManualHeightDown						:BOOL;  					// Na dół

	//Chwytak zakrecarki szczękowej
	lrGripperScrewerCatchHeightCV						:LREAL;  					// Aktualna pozycja
	bGripperScrewerCatchHeightSet						:BOOL;						// Ustaw
    bGripperScrewerCatchManualUp						:BOOL;  					// Do góry
    bGripperScrewerCatchManualDown						:BOOL;  					// Na dół

	//Chwytak 1
	iGripperScrewerCatch1State							:INT;						// Stan
	sGripperScrewerCatch1State							:STRING;					// Stan
	bGripperScrewerCatch1ManualActuator					:BOOL;  					// Chwytak
	//chwytak 2
	iGripperScrewerCatch2State							:INT;						// Stan
	sGripperScrewerCatch2State							:STRING;                    // Stan
	bGripperScrewerCatch2ManualActuator					:BOOL;  					// Chwytak
	//Stoper
	bGripperScrewerStoperManualActuator					: BOOL;
		
	
	(*****P11_CapCorrectCheck********) 
	//Sprawdzanie zakręcenia                  			
	iCapCorrectCheckState								:INT;         				// Stan
	sCapCorrectCheckState								:STRING;         			// Stan
    bCapCorrectCheckHoming								:BOOL;					   	// Bazowanie
    bCapCorrectCheckIgnoreErrors						:BOOL;				    	// Ignoruj błędy
   	lrCapCorrectCheckHeightCV							:LREAL;				 		// Aktualna wysokość
    bCapCorrectCheckManualHeightUp						:BOOL; 						// Do góry
    bCapCorrectCheckManualHeightDown					:BOOL;			 			// Na dół
	bCapCorrectCheckHeightSet							:BOOL;						// Ustaw
	AsCapCorrectCheckCameraProgramDescription			:ARRAY [0..10] OF STRING;	// Opis programów kamer, 0 - Opis programu nr 1, 1 - Opis programu nr 2
	bCapCorrectCheckCameraOK							:BOOL;						// Orientacja nasadki OK
                               			
	(*****P13_BottleTransfer********)
	//Przenoszenie butelek
	iBottleTransferState								:INT; 						// Stan
	sBottleTransferState								:STRING;                    // Stan      
	bBottleTransferHoming								:BOOL;  					// Bazowanie 
	bBottleTransferHeightSet 							:BOOL;			 			// Ustaw
	bBottleTransferIgnoreErrors							:BOOL; 						// Ignoruj błedy
	bBottleTransferRun									:BOOL; 						// Cykl Pobierz
    bBottleTransferPlace								:BOOL; 						// Cykl Odłóż
    nBottleTransferPlaceOption							:INT; 					  	// Miejsce odłozenia	(1 - etykieciarka, 2 - odrzut)
	nBottleTransferPickOption							:INT;						// Miejsce pobrania		(1- 1 butelka, 2 - 2 butelki)
	bBottleTransferManualCatch							:BOOL;					 	// Chwytak
    bBottleTransferManualPick							:BOOL; 						// Pobierz 1 but.
	bBottleTransferManualPick2 							:BOOL; 						// Pobierz 2 but.
    bBottleTransferManualPlace1							:BOOL; 						// Odłóż na etykieciarkę
    bBottleTransferManualPlace2							:BOOL; 						// Odłóż na odrzut
    bBottleTransferManualReadyPosition					:BOOL; 						// Gotowość
	bBottleTransferManualStartInkJet					:BOOL; 						// Start InkJet
	bBottleTransferManualStopInkJet						:BOOL; 						// Stop InkJet
	bBottleTransferManualWeight							:BOOL;						// Waga
	bBottleTransferManualEditOffset						:BOOL; 						// Edycja offsetów		
	bBottleTransferAllFormsToLabeler					:BOOL;						// Przekładanie wszystkich na etykieciarkę (opis na głównym: "Przenoszenie wszystkich butelek na etykieciarke") (Umieścić na ekranie głównym)
	bBottleTransferAllFormsToExit						:BOOL;						// Przekadanie wszystkich na odrzut (opis na głównym: "Przenoszenie wszystkich butelek na etykieciarke") (Umieścić na ekranie głównym)
	bBottleTransferLubricationReset						:BOOL;						// Reset smarowania
	aBottleTransferLoadAxis								:ARRAY[0..3] OF INT;		// [H] Aktualne obciążenia osi J1 J2 J3 J4	 
	iBottleTransferLock									:INT;						// Blokowanie przycisków trybu manualnego (b0-1 blokuj 
	bBottleTransferForceWeight							:BOOL;						// Przesuń następne opakowanie na wagę																					// 2#11111111 - nie moge nic  
																					// 2#11111110 - moge pobrać (tylko Pick1 i Pick 2 odblokowane)
																					// 2#11101001 - moge odłożyć, odrzucić i pojechać przed inkjet		
																					// 2#11110111 - moge jechać tylko do gotowości
																					// 2#11110111 - moge jechać tylko do gotowości
																					// 2#11011111 - moge jechać do koniec inkjet
																					// 2#10101101 - moge odłożyć na ety., wrocić przed inkjet
																					// 2#11111110 - moge pobrać

	(*Wersja 2, jeżeli nie uda się odtworzyć widoczności po zmiennej..Lock'	*)																				
	bBottleTransferManualCatchVisibility				:BOOL;					 	// Chwytak - przycisk odblokowany
    bBottleTransferManualPickVisibility					:BOOL; 						// Pobierz 1 but. - przycisk odblokowany
	bBottleTransferManualPick2Visibility 				:BOOL; 						// Pobierz 2 but. - przycisk odblokowany
    bBottleTransferManualPlace1Visibility				:BOOL; 						// Odłóż na etykieciarkę - przycisk odblokowany
    bBottleTransferManualPlace2Visibility				:BOOL; 						// Odłóż na odrzut - przycisk odblokowany
    bBottleTransferManualReadyPositionVisibility		:BOOL; 						// Gotowość - przycisk odblokowany
	bBottleTransferManualStartInkJetVisibility			:BOOL; 						// Start InkJet - przycisk odblokowany
	bBottleTransferManualStopInkJetVisibility			:BOOL; 						// Stop InkJet - przycisk odblokowany

	(*****P13_BottleTransferAfterDrag********)
	//Przeciąganie formatek 
	iBottleTransferAfterDragState						:INT;						// Stan
	sBottleTransferAfterDragState						:STRING;					// Stan
	bBottleTransferAfterDragRun							:BOOL;						// Cykl
	bBottleTransferAfterDragHoming						:BOOL;						// Bazowanie 
	bBottleTransferAfterDragIgnoreError					:BOOL;						// Ignoruj błędy
	bBottleTransferAfterDragManualActuator					:BOOL;						// Podnosnik
	//Stoper,szlaban
	bBottleTransferAfterDragManualStoper				:BOOL;						// Stoper
	bBottleTransferAfterDragManualGate					:BOOL;						// Stoper

	
	(*****P14_BadBottleConyevor********)
	//Transporter odzutu
	iBadBottleConveyorState								:INT; 					 	// Stan
	sBadBottleConveyorState								:STRING; 					// Stan
	nBadBottleConveyorCV								:UDINT; 					// Aktualna prędkość [rpm]
	bBadBottleConveyorManualCmdStart					:BOOL; 						// Start 
	bBadBottleConveyorManualDirection 					:BOOL; 						// Kierunek
	
	(*******P14_TurnTable********)
	
	(********P15_FormTransporters********)
	//Transporter przed dozownikami
	iFormTransporterDispencerState						:INT; 					 	// Stan
	sFormTransporterDispencerState						:STRING; 					// Stan
	nFormTransporterDispencerVelocityCV					:INT;						// Aktualna prędkość
	bFormTransporterDispencerManualCmdStart				:BOOL; 					 	// Start
	//Transporter za dozownikami
	iFormTransporterScrewerState						:INT; 					 	// Stan
	sFormTransporterScrewerState						:STRING; 					// Stan
	nFormTransporterScrewerVelocityCV					:INT;						// Aktualna prędkość
	bFormTransporterScrewerManualCmdStart				:BOOL; 					 	// Start
	//Transporter przed zakręcarką
	iFormTransporterBeforeScrewerState					:INT;						// Stan
	sFormTransporterBeforeScrewerState					:STRING;					// Stan
	nFormTransporterBeforeScrewerVelocityCV				:INT;						// Aktualna prędkość
	bFormTransporterBeforeScrewerManualCmdStart			:BOOL; 						// Start
	//Spowalniacz
	iFormTransporterAfterCapSorterState							:INT;						// Stan pracy spowalniacz formatek
	sFormTransporterAfterCapSorterState							:STRING;					// Stan pracy spowialniacza formatek
	nFormTransporterAfterCapSorterVelocityCV					:INT;						// Aktualna predkosc spowalniacza
	bFormTransporterAfterCapSorterManualCmdStart				:BOOL; 						// Stan pracy spowalniacza formatek
	//Transporter za zakręcarką
	iFormTransporterAfterScreweArState					:INT;						// Stan
	sFormTransporterAfterScrewerState					:STRING;					// Stan
	nFormTransporterAfterScrewerVelocityCV				:INT;						// Aktualna prędkość
	bFormTransporterAfterScrewerManualCmdStart			:BOOL; 						// Start

	(*****P16_LabelMachine********)
	//Etykieciarka
	bLabelMachine1ManualStart 							:BOOL;						// Start
	
	(*****P17_CircularInkJet********)
	//[H] Inkjet obrotowy
	bCircularInkjetRollersManualStart 					:BOOL;						// [H] Rolki
	bCircularInkjetActuatorManualStart 					:BOOL;						// [H] Chwytak
	(*****P17_TurnTables********)
	//Stół odbiorczy
	bExitTurnTable1ManualStart 							:BOOL;						// Start
	bExitTurnTableManualActuator						:BOOL;						// Siłownik stołu odbiorczego
	//Transporter odbiorczy
	bExitConveyorManualStart							:BOOL;						// Transporter
	bExitConveyorGateManualActuator						:BOOL;						// Szlaban transportera odbiorczego
	
	(*****P20_ExhaustFan*****)
	//Wentylator Ex
	iExhaustFanState									:INT;						// Stan
	sExhaustFanState									:STRING;					// Stan
	udiExhaustFanVelocityCV								:UDINT;						// Aktualna prędkość wentylatora
	bExhaustFanManualCmdStart							:BOOL;						// Start
	
	
	bOffPLC			:BOOL;					//sygnał do wyłączenia PLC
	UPPackMLState 	:INT;					//statusy PckML kartoniarki
	EPPackMLState	:INT;					//statusy PckML paletyzatora
	
	//Zmienne do odczytu prądu krokówek
	DCcurrertStepeerScrewers AT%I*:UINT;     
	DCcurrertStepeerDosers AT%I*:UINT;
	
	
	
(********************************************************************************************************************************************)
(********************************************************************************************************************************************)

	(******* Zmienne do receptury*********)

	(*****P00_Recipes***) 
	(*****Receptury****)	
	bChooseRecipe										:BOOL; 						// Wczytaj
	bRecipeLoading 										:BOOL; 						// Trwa wczytywanie
	
	sRecipeNameShow										:WSTRING;		//	P030_Recipes.stActRecipe.stUBL.sRecipeNameShow;		// Nazwa 
	sRecipeDescriptionShow								:WSTRING(1000);	//	P030_Recipes.stActRecipe.stUBL.sRecipeDescriptionShow;		// Nazwa
	sRecipeDispencerDescriptionShow						:WSTRING(250);		
	sRecipeCapsDescriptionShow 							:WSTRING(250);				
	sRecipeFormersDescriptionShow                       :WSTRING(250);
	sRecipeRobotDescriptionShow                         :WSTRING(250);
	sRecipeBottleSorterDescriptionShow                  :WSTRING(250);
	sRecipeCapSorterDescriptionShow                     :WSTRING(250);
	sRecipeCapPutterDescriptionShow                     :WSTRING(250);
                                                                        //
	sRecipeIndexShow									:STRING;		//	P030_Recipes.stActRecipe.stUBL.sRecipeIndexShow;		// Indeks 
	nRecipeIndexShow									:REAL;			//	P030_Recipes.stActRecipe.stUBL.nRecipeIndexShow;		// Indeks 
                                                                        //
	//Parametry opakowania
 	iPackagePuckInsertHeightShow						:INT; 			// Wysokość wkładki w formatce (0-100mm)                
	iPackageMassTypeShow								:INT; 			// Typ masy (0-Woda, 1-Olej, 2-Mydło, 3-Krem itd.)
	iPackageCapTypeShow									:INT; 			// Typ nasadki (0-Fliptop, 1-Pompka/Atomizer, 2-Fliptop z boku, 3-Airless, 4-Deko z boku, 5- Deko
	iPackageCapDiameterShow								:INT;			// Średnica nasadki (5-50mm),
	iPackageHeightShow									:INT;			// Wysokość butelki (50-300mm),
	iPackageCappedHeightShow							:INT;			// Wysokość butelki razem z dokręconą nakrętką i formatką (50-350mm),	
	iPackageNozzleDiameterShow							:INT;			// Srednica wylewki (6-30mm),	
	                                                                        //
	//[H] Praca w trybie wybuchowym                                     //
	bExEnableShow										:BOOL;			//	P030_Recipes.stActRecipe.stUBL.bExEnableShow;		// [H] Tryb EX
	                                                                    //
	// Podajnik butelek  	                                            //
	bBottleFeederEnableShow								:BOOL;   		//	P030_Recipes.stActRecipe.stUBL.bBottleFeederEnableShow							 		// Aktywacja
	iBottleFeederTurntableVelocitySVShow				:UDINT;			//	P030_Recipes.stActRecipe.stUBL.iBottleFeederTurntableVelocitySVShow	// Prędkość stołu
	iBottleFeederBottleSensorDelayShow					:INT;			//	P030_Recipes.stActRecipe.stUBL.iBottleFeederBottleSensorDelayShow		// Opóźnienie wjazdu butelki
	iBottleFeederFormGateDelayShow						:INT;			//	P030_Recipes.stActRecipe.stUBL.iBottleFeederFormGateDelayShow			// Czas otwarcia szlabanu formatek
	iBottleFeederAllowFormDelayShow						:INT;			//	P030_Recipes.stActRecipe.stUBL.iBottleFeederAllowFormDelayShow			// Czas po którym formatka zostaje wypuszczona bez butelki
                                                                        //
	// Podajnik opakowań	                                            //
	bPucksInserterEnableShow							:BOOL;   		//	P030_Recipes.stActRecipe.stUBL.bPucksInserterEnableShow						// Aktywacja
	iPucksInserterTurntableVelocitySVShow				:UDINT;			//	P030_Recipes.stActRecipe.stUBL.iPucksInserterTurntableVelocitySVShow			// Prędkość stołu
	iPucksInserterConveyorVelocitySVShow				:UDINT;			//	P030_Recipes.stActRecipe.stUBL.iPucksInserterConveyorVelocitySVShow			// Prędkość transportera
	iPucksInserterBottleSensorDelayShow					:INT;			//	P030_Recipes.stActRecipe.stUBL.iPucksInserterBottleSensorDelayShow				// Opóźnienie wjazdu butelki
	iPucksInserterFormGateDelayShow						:INT;			//	P030_Recipes.stActRecipe.stUBL.iPucksInserterFormGateDelayShow					// Czas otwarcia szlabanu formatek
	iPucksInserterAllowFormDelayShow					:INT;			//	P030_Recipes.stActRecipe.stUBL.iPucksInserterAllowFormDelayShow				// Czas po którym formatka zostaje wypuszczona bez butelki
	lrPucksInserterWheelOffsetShow						:LREAL;			//	P030_Recipes.stActRecipe.stUBL.lrPucksInserterWheelOffsetShow					// Offset karuzeli +-10 st.
	lrPucksInserterWheelAccelerationShow				:LREAL;			//	P030_Recipes.stActRecipe.stUBL.lrPucksInserterWheelAccelerationShow			// Przyspieszenie 
	lrPucksInserterWheelVelocityShow					:LREAL;			//	P030_Recipes.stActRecipe.stUBL.lrPucksInserterWheelVelocityShow				// Prędkość 
	lrPucksInserterHammerHeightSVShow					:LREAL;  		//	P030_Recipes.stActRecipe.stUBL.lrPucksInserterHammerHeightSVShow				// Zadana wysokość
	                                                                    //                                                                                    									
	//Vasyl 27.05 Stół podający butelki                                 //                                               									
	udiPucksInserterPushTableVelocityShow				:UDINT;			//	P030_Recipes.stActRecipe.stUBL.udiPucksInserterPushTableVelocityShow			 									
	iPucksInserterPushTableRollersVelocityShow			:INT;           //  P030_Recipes.stActRecipe.stUBL.iPucksInserterPushTableRollersVelocityShow		 									
	udiPucksInserterPushTableActuatorPUSHDelayShow		:UDINT;         //  P030_Recipes.stActRecipe.stUBL.udiPucksInserterPushTableActuatorPUSHDelayShow	 									
	udiPucksInserterPushTableActuatorPULLDelayShow		:UDINT;         //  P030_Recipes.stActRecipe.stUBL.udiPucksInserterPushTableActuatorPULLDelayShow	 									
	bPucksInserterPushTableActuatorEnableShow			:BOOL;          //  P030_Recipes.stActRecipe.stUBL.bPucksInserterPushTableActuatorEnableShow		 									
	bPucksInserterPushTableRollerEnableShow				:BOOL;          //  P030_Recipes.stActRecipe.stUBL.bPucksInserterPushTableRollerEnableShow			 									
	bPucksInserterPushTableEnableShow					:BOOL;          //  P030_Recipes.stActRecipe.stUBL.bPucksInserterPushTableEnableShow				 	
	udiPucksInserterPushTableOFFDelayShow				:UDINT;			//	P030_Recipes.stActRecipe.stUBL.udiPucksInserterPushTableOFFDelayShow					
	                                                                    //
	                                                                    //
	//Sorter butelek                                                    //
	//Parametry receptur z innego sterownika                            //
	                                                                    //
	//[H] Parametry szlabanów                                           //
	bGateBeforeDispencersEnableShow						:BOOL;			//	P030_Recipes.stActRecipe.stUBL.bGateBeforeDispencersEnableShow									// [H] Aktywacja
	nGateBeforeDispencersTimeFormInsertingShow			:UINT;			//	P030_Recipes.stActRecipe.stUBL.nGateBeforeDispencersTimeFormInsertingShow						// [H] Czas wyjazdu formatki	
	bGateAfterWeightEnableShow							:BOOL;			//	P030_Recipes.stActRecipe.stUBL.bGateAfterWeightEnableShow										// [H] Aktywacja
	nGateAfterWeightTimeFormInsertingShow				:UINT;			//	P030_Recipes.stActRecipe.stUBL.nGateAfterWeightTimeFormInsertingShow							// [H] Czas wyjazdu formatki
	bGateRobotEnableShow								:BOOL;			//	P030_Recipes.stActRecipe.stUBL.bGateRobotEnableShow											// [H] Aktywacja
	nGateRobotTimeFormInsertingShow						:UINT;			//	P030_Recipes.stActRecipe.stUBL.nGateRobotTimeFormInsertingShow									// [H] Czas przejazdu formatki
                                                                        //                                        										
	//Przeciaganie formatek pod dozownikami	lewe                        //                                        										
	bFormsDragingLeftEnableShow							:BOOL;			//	P030_Recipes.stActRecipe.stUBL.bFormsDragingLeftEnableShow								// Aktywacja
	lrFormsDragingLeftVelocityShow						:LREAL; 		//	P030_Recipes.stActRecipe.stUBL.lrFormsDragingLeftVelocityShow							// Prędkość [mm/s] (100-1000)
 	lrFormsDragingLeftAccelerationShow					:LREAL;			//	P030_Recipes.stActRecipe.stUBL.lrFormsDragingLeftAccelerationShow					// Przyspieszenie [mm/s2] (100-10000)
	lrFormsDragingLeftDecelerationShow					:LREAL;			//	P030_Recipes.stActRecipe.stUBL.lrFormsDragingLeftDecelerationShow					// Hamowanie [mm/s2] (100-10000)
	//Przeciaganie formatek pod dozownikami	prawe	                    //                                        										
	bFormsDragingRightEnableShow						:BOOL;			//	P030_Recipes.stActRecipe.stUBL.bFormsDragingRightEnableShow							// Aktywacja
	lrFormsDragingRightVelocityShow						:LREAL; 		//	P030_Recipes.stActRecipe.stUBL.lrFormsDragingRightVelocityShow							// Prędkość [mm/s] (100-1000)   
 	lrFormsDragingRightAccelerationShow					:LREAL;			//	P030_Recipes.stActRecipe.stUBL.lrFormsDragingRightAccelerationShow						// Przyspieszenie [mm/s2] (100-1
	lrFormsDragingRightDecelerationShow					:LREAL;			//	P030_Recipes.stActRecipe.stUBL.lrFormsDragingRightDecelerationShow						// Hamowanie [mm/s2] (100-10000)
	                                                                    //                                        												
	//Dozowniki                                                         //                                        												
	bDosingTwoPhasesShow								:BOOL;			//	P030_Recipes.stActRecipe.stUBL.bDosingTwoPhasesShow																			// Dozowanie dwu-fazowe
    lrDispencersLifterReadyPositionShow					:LREAL;			//	P030_Recipes.stActRecipe.stUBL.lrDispencersLifterReadyPositionShow																// Pozycja gototości 
	uiDispencerStartDosingDelayShow						:UINT;			//	P030_Recipes.stActRecipe.stUBL.uiDispencerStartDosingDelayShow																	// Zwłoka rozpoczęcia dozowania
	bDispencer1EnableShow								:BOOL; 			//	P030_Recipes.stActRecipe.stUBL.bDispencer1EnableShow								// Aktywacja dozownika 1                                                        				
	bDispencer2EnableShow								:BOOL; 			//	P030_Recipes.stActRecipe.stUBL.bDispencer2EnableShow								// Aktywacja dozownika 2 
	bDispencer3EnableShow								:BOOL; 			//	P030_Recipes.stActRecipe.stUBL.bDispencer3EnableShow								// Aktywacja dozownika 3  
	bDispencer4EnableShow								:BOOL; 			//	P030_Recipes.stActRecipe.stUBL.bDispencer4EnableShow								// Aktywacja dozownika 4  
	                                                                    //
	//Dozownik 12 (druga faza)                                       	//			
	lrDispencer1DoseVolumeShow							:LREAL:=300; 	//	P030_Recipes.stActRecipe.stUBL.lrDispencer1DoseVolumeShow						// Objętość do wydozowania [ml]
	lrDispencer1Phase1VolumeShow						:LREAL:=100;	//	P030_Recipes.stActRecipe.stUBL.lrDispencer1Phase1VolumeShow					// Objętość fazy początkowej [ml]
	lrDispencer1Phase2VolumeShow						:LREAL:=200;	//	P030_Recipes.stActRecipe.stUBL.lrDispencer1Phase2VolumeShow					// Objętość fazy końcowej [ml]
	lrDispencer1Phase1VelocityShow						:LREAL:=500;	//	P030_Recipes.stActRecipe.stUBL.lrDispencer1Phase1VelocityShow					// Prędkość fazy początkowej [ml/s]
	lrDispencer1Phase2VelocityShow						:LREAL:=500;	//	P030_Recipes.stActRecipe.stUBL.lrDispencer1Phase2VelocityShow					// Prędkość fazy dozowania [ml/s]
	lrDispencer1Phase3VelocityShow						:LREAL:=500;	//	P030_Recipes.stActRecipe.stUBL.lrDispencer1Phase3VelocityShow					// Prędkość fazy koncowej [ml/s]
	lrDispencer1SuckVelocityShow						:LREAL:=500;	//	P030_Recipes.stActRecipe.stUBL.lrDispencer1SuckVelocityShow					// Prędkość zasysania masy [ml/s2]
	lrDispencer1Phase1AccelerationShow					:LREAL:=3000;	//	P030_Recipes.stActRecipe.stUBL.lrDispencer1Phase1AccelerationShow				// Przyśpieszenie fazy początkowej [ml/s2]
	lrDispencer1Phase2AccelerationShow					:LREAL:=3000;	//	P030_Recipes.stActRecipe.stUBL.lrDispencer1Phase2AccelerationShow				// Przyśpieszenie fazy dozowania [ml/s2]
	lrDispencer1Phase3AccelerationShow					:LREAL:=3000;	//	P030_Recipes.stActRecipe.stUBL.lrDispencer1Phase3AccelerationShow				// Przyśpieszenie fazy końcowej [ml/s2]
	lrDispencer1SuckAccelerationShow					:LREAL:=3000;	//	P030_Recipes.stActRecipe.stUBL.lrDispencer1SuckAccelerationShow				// Przyśpieszenie zasysania masy [ml/s2]
	lrDispencer1Phase1DecelerationShow					:LREAL:=3000;	//	P030_Recipes.stActRecipe.stUBL.lrDispencer1Phase1DecelerationShow				// Dynamika zwalniania w fazie początkowej
	lrDispencer1Phase2DecelerationShow					:LREAL:=3000;	//	P030_Recipes.stActRecipe.stUBL.lrDispencer1Phase2DecelerationShow				// Dynamika zwalniania dozowania
	lrDispencer1Phase3DecelerationShow					:LREAL:=3000;	//	P030_Recipes.stActRecipe.stUBL.lrDispencer1Phase3DecelerationShow				// Dynamika zwalniania fazy końcowej
	udiDispencer1DosingDoneDelayTimeShow				:UDINT:=0; 		//	P030_Recipes.stActRecipe.stUBL.udiDispencer1DosingDoneDelayTimeShow			// Zwłoka po wydozowaniu
	lrDispencer1SuckValveOpenVolumeShow					:LREAL:=0;		//	P030_Recipes.stActRecipe.stUBL.lrDispencer1SuckValveOpenVolumeShow				// Objętość przy której otwiera się zawór ssania [3] 
	lrDispencer1SuckValveOpenTimeDelayShow				:LREAL:=0;		//	P030_Recipes.stActRecipe.stUBL.lrDispencer1SuckValveOpenTimeDelayShow			// Zwłoka rozpoczęcia ssania po tłoczeniu [ms] [3]
	lrDispencer1SuckValveCloseVolumeShow				:LREAL:=0;		//	P030_Recipes.stActRecipe.stUBL.lrDispencer1SuckValveCloseVolumeShow			// [H] Objętość zamknięcia zaworu ssania od końca ssania [4]
	lrDispencer1SuckValveCloseTimeDelayShow				:LREAL:=0;		//	P030_Recipes.stActRecipe.stUBL.lrDispencer1SuckValveCloseTimeDelayShow			// Zwłoka zamknięcia zaworu ssącego [ms] [4] 
	lrDispencer1DoseValveOpenVolumeShow					:LREAL:=0;		//	P030_Recipes.stActRecipe.stUBL.lrDispencer1DoseValveOpenVolumeShow				// [H] Objętość przy której otwiera się zawór tłoczenia [ml] [1]
	lrDispencer1DoseValveOpenTimeAccShow				:LREAL:=0;		//	P030_Recipes.stActRecipe.stUBL.lrDispencer1DoseValveOpenTimeAccShow			// Wyprzedzenie otwarcia zaworu tłoczenia [1] [ms]
	lrDispencer1DoseValveCloseVolumeShow				:LREAL:=0;		//	P030_Recipes.stActRecipe.stUBL.lrDispencer1DoseValveCloseVolumeShow			// Pozostała objętość dozy - zamknięcie zaworu tłoczenia [ml] [2]
	lrDispencer1DoseValveCloseTimeDecShow				:LREAL:=0;		//	P030_Recipes.stActRecipe.stUBL.lrDispencer1DoseValveCloseTimeDecShow			// Zwłoka zamkniecia zaworu tłoczenia [2] [ms]
	lrDispencer1DoseSuckingVolumeShow					:LREAL:=0;		//	P030_Recipes.stActRecipe.stUBL.lrDispencer1DoseSuckingVolumeShow				// Ilość dozy do posysenia [ml]	[5] [Podsysanie] 
	lrDispencer1DoseSuckingTimeDelayShow				:LREAL:=0;		//	P030_Recipes.stActRecipe.stUBL.lrDispencer1DoseSuckingTimeDelayShow			// Opóźnienie podsysania [ms] [6] [Podsysanie] 
	bDispencer1DoseSuckingShow							:BOOL;			//	P030_Recipes.stActRecipe.stUBL.bDispencer1DoseSuckingShow						// Aktywacja podsysania
	bDispencer1LiftSynchroPh1Show						:BOOL;			//	P030_Recipes.stActRecipe.stUBL.bDispencer1LiftSynchroPh1Show					// Synchronizacja z podnosnikiem w fazie początkowej
	bDispencer1LiftSynchroPh2Show						:BOOL; 			//	P030_Recipes.stActRecipe.stUBL.bDispencer1LiftSynchroPh2Show					// Synchronizacja z podnosnikiem w fazie dozowania
	bDispencer1LiftSynchroPh3Show						:BOOL; 			//	P030_Recipes.stActRecipe.stUBL.bDispencer1LiftSynchroPh3Show					// Synchronizacja z podnosnikiem w fazie końcowej
	lrDispencer1LifterStartDosePositionShow				:LREAL:=20;		//	P030_Recipes.stActRecipe.stUBL.lrDispencer1LifterStartDosePositionShow			// Pozycja rozpoczęcia dozowania
	lrDispencer1LifterStopDosePositionShow				:LREAL:=60;		//	P030_Recipes.stActRecipe.stUBL.lrDispencer1LifterStopDosePositionShow			// Pozycja zakończenia dozowania
	lrDispencer1LifterVelocityShow						:LREAL:=100;	//	P030_Recipes.stActRecipe.stUBL.lrDispencer1LifterVelocityShow					// [H] Prędkość podnośnika 
	lrDispencer1LifterAccelerationShow					:LREAL:=2;		//	P030_Recipes.stActRecipe.stUBL.lrDispencer1LifterAccelerationShow				// [H] Przyspieszenie podnośnika
	lrDispencer1LifterDecelerationShow					:LREAL:=2;		//	P030_Recipes.stActRecipe.stUBL.lrDispencer1LifterDecelerationShow				// [H] Zwalnianie podnośnika
                                                                        //
	//Dozowniki 34 (pierwsza faza)                                      //       				
    lrDispencer2DoseVolumeShow							:LREAL:=300; 	//	P030_Recipes.stActRecipe.stUBL.lrDispencer2DoseVolumeShow						// Objętość do wydozowania                                           
	lrDispencer2Phase1VolumeShow						:LREAL:=100;	//	P030_Recipes.stActRecipe.stUBL.lrDispencer2Phase1VolumeShow					// Objętość fazy początkowej                                         
	lrDispencer2Phase2VolumeShow						:LREAL:=200;	//	P030_Recipes.stActRecipe.stUBL.lrDispencer2Phase2VolumeShow					// Objętość fazy końcowej                                            
	lrDispencer2Phase1VelocityShow						:LREAL:=500;	//	P030_Recipes.stActRecipe.stUBL.lrDispencer2Phase1VelocityShow					// Prędkość fazy początkowej                                         
	lrDispencer2Phase2VelocityShow						:LREAL:=500;	//	P030_Recipes.stActRecipe.stUBL.lrDispencer2Phase2VelocityShow					// Prędkość fazy dozowania                                           
	lrDispencer2Phase3VelocityShow						:LREAL:=500;	//	P030_Recipes.stActRecipe.stUBL.lrDispencer2Phase3VelocityShow					// Prędkość fazy koncowej                                            
	lrDispencer2SuckVelocityShow						:LREAL:=500;	//	P030_Recipes.stActRecipe.stUBL.lrDispencer2SuckVelocityShow					// Prędkość zasysania masy                                           
	lrDispencer2Phase1AccelerationShow					:LREAL:=3000;	//	P030_Recipes.stActRecipe.stUBL.lrDispencer2Phase1AccelerationShow				// Przyspieszenie fazy początkowej                                   
	lrDispencer2Phase2AccelerationShow					:LREAL:=3000;	//	P030_Recipes.stActRecipe.stUBL.lrDispencer2Phase2AccelerationShow				// Przyspieszenie fazy dozowania                                     
	lrDispencer2Phase3AccelerationShow					:LREAL:=3000;	//	P030_Recipes.stActRecipe.stUBL.lrDispencer2Phase3AccelerationShow				// Przyspieszenie fazy końcowej                                      
	lrDispencer2SuckAccelerationShow					:LREAL:=3000;	//	P030_Recipes.stActRecipe.stUBL.lrDispencer2SuckAccelerationShow				// Przyspieszenie zasysania masy                                     
	lrDispencer2Phase1DecelerationShow					:LREAL:=3000;	//	P030_Recipes.stActRecipe.stUBL.lrDispencer2Phase1DecelerationShow				// Dynamika zwalniania w fazie początkowej                           
	lrDispencer2Phase2DecelerationShow					:LREAL:=3000;	//	P030_Recipes.stActRecipe.stUBL.lrDispencer2Phase2DecelerationShow				// Dynamika zwalniania dozowania                                     
	lrDispencer2Phase3DecelerationShow					:LREAL:=3000;	//	P030_Recipes.stActRecipe.stUBL.lrDispencer2Phase3DecelerationShow				// Dynamika zwalniania fazy końcowej                                 
	udiDispencer2DosingDoneDelayTimeShow				:UDINT:=0; 		//	P030_Recipes.stActRecipe.stUBL.udiDispencer2DosingDoneDelayTimeShow			// Zwłoka po wydozowaniu                                             
	lrDispencer2SuckValveOpenVolumeShow					:LREAL:=0;		//	P030_Recipes.stActRecipe.stUBL.lrDispencer2SuckValveOpenVolumeShow				// Objętość przy której otwiera się zawór ssania [3]                 
	lrDispencer2SuckValveOpenTimeDelayShow				:LREAL:=0;		//	P030_Recipes.stActRecipe.stUBL.lrDispencer2SuckValveOpenTimeDelayShow			// Zwłoka rozpoczęcia ssania po tłoczeniu [ms] [3]                   
	lrDispencer2SuckValveCloseVolumeShow				:LREAL:=0;		//	P030_Recipes.stActRecipe.stUBL.lrDispencer2SuckValveCloseVolumeShow			// [H] Objętość zamknięcia zaworu ssania od końca ssania [4]    
	lrDispencer2SuckValveCloseTimeDelayShow				:LREAL:=0;		//	P030_Recipes.stActRecipe.stUBL.lrDispencer2SuckValveCloseTimeDelayShow			// Zwłoka zamknięcia zaworu ssącego [ms] [4]                         
	lrDispencer2DoseValveOpenVolumeShow					:LREAL:=0;		//	P030_Recipes.stActRecipe.stUBL.lrDispencer2DoseValveOpenVolumeShow				// [H] Objętość przy której otwiera się zawór tłoczenia [ml] [1]
	lrDispencer2DoseValveOpenTimeAccShow				:LREAL:=0;		//	P030_Recipes.stActRecipe.stUBL.lrDispencer2DoseValveOpenTimeAccShow			// Wyprzedzenie otwarcia zaworu tłoczenia [1] [ms]                   
	lrDispencer2DoseValveCloseVolumeShow				:LREAL:=0;		//	P030_Recipes.stActRecipe.stUBL.lrDispencer2DoseValveCloseVolumeShow			// Pozostała objętość dozy - zamknięcie zaworu tłoczenia [ml] [2]    
	lrDispencer2DoseValveCloseTimeDecShow				:LREAL:=0;		//	P030_Recipes.stActRecipe.stUBL.lrDispencer2DoseValveCloseTimeDecShow			// Zwłoka zamkniecia zaworu tłoczenia [2] [ms]                       
	lrDispencer2DoseSuckingVolumeShow					:LREAL:=0;		//	P030_Recipes.stActRecipe.stUBL.lrDispencer2DoseSuckingVolumeShow				// Ilość dozy do posysenia [ml]	[5] [Podsysanie]                     
	lrDispencer2DoseSuckingTimeDelayShow				:LREAL:=0;		//	P030_Recipes.stActRecipe.stUBL.lrDispencer2DoseSuckingTimeDelayShow			// Opóźnienie podsysania [ms] [6] [Podsysanie]                       
	bDispencer2DoseSuckingShow							:BOOL;			//	P030_Recipes.stActRecipe.stUBL.bDispencer2DoseSuckingShow						// Aktywacja podsysania                                              
	bDispencer2LiftSynchroPh1Show						:BOOL;			//	P030_Recipes.stActRecipe.stUBL.bDispencer2LiftSynchroPh1Show					// Synchronizacja z podnosnikiem w fazie początkowej                 
	bDispencer2LiftSynchroPh2Show						:BOOL; 			//	P030_Recipes.stActRecipe.stUBL.bDispencer2LiftSynchroPh2Show					// Synchronizacja z podnosnikiem w fazie dozowania                   
	bDispencer2LiftSynchroPh3Show						:BOOL; 			//	P030_Recipes.stActRecipe.stUBL.bDispencer2LiftSynchroPh3Show					// Synchronizacja z podnosnikiem w fazie końcowej                    
	lrDispencer2LifterStartDosePositionShow				:LREAL:=20;		//	P030_Recipes.stActRecipe.stUBL.lrDispencer2LifterStartDosePositionShow			// Pozycja rozpoczęcia dozowania                                     
	lrDispencer2LifterStopDosePositionShow				:LREAL:=60;		//	P030_Recipes.stActRecipe.stUBL.lrDispencer2LifterStopDosePositionShow			// Pozycja zakończenia dozowania                                     
	lrDispencer2LifterVelocityShow						:LREAL:=100;	//	P030_Recipes.stActRecipe.stUBL.lrDispencer2LifterVelocityShow					// [H] Prędkość podnośnika                                      
	lrDispencer2LifterAccelerationShow					:LREAL:=2;		//	P030_Recipes.stActRecipe.stUBL.lrDispencer2LifterAccelerationShow				// [H] Przyspieszenie podnośnika                                
	lrDispencer2LifterDecelerationShow					:LREAL:=2;		//	P030_Recipes.stActRecipe.stUBL.lrDispencer2LifterDecelerationShow				// [H] Zwalnianie podnośnika                                    
                                                            		    //
	//Chwytak dozowników 1234                                           //
	bDispencersCatchEnableShow	      					:BOOL;			//	P030_Recipes.stActRecipe.stUBL.bDispencersCatchEnableShow	      			// [H] Aktywacja    
 	bDispencersCatchMaxPressureShow	      				:BOOL;			//	P030_Recipes.stActRecipe.stUBL.bDispencersCatchMaxPressureShow	    		// Zwiększona siła chwytania            		
	lrDispencersCatchHeightSVShow						:LREAL:=86;  	//	P030_Recipes.stActRecipe.stUBL.lrDispencersCatchHeightSVShow				// Pozycja chwytaka
 	//Kalibracja chwytaków 1234                                         //
    lrDispencersCatch1ClosedValueShow                   :LREAL;         //  P030_Recipes.stActRecipe.stUBL.lrDispencersCatch1ClosedValueShow        // Chwytak 1 | wartość kalibracji zamkniętego chwytaka
    lrDispencersCatch1OpenValueShow                     :LREAL;         //  P030_Recipes.stActRecipe.stUBL.lrDispencersCatch1OpenValueShow           // Chwytak 1 | wartość kalibracji otwartego chwytaka
    lrDispencersCatch2ClosedValueShow                   :LREAL;         //  P030_Recipes.stActRecipe.stUBL.lrDispencersCatch2ClosedValueShow         // Chwytak 2 | wartość kalibracji zamkniętego chwytaka
    lrDispencersCatch2OpenValueShow                     :LREAL;         //  P030_Recipes.stActRecipe.stUBL.lrDispencersCatch2OpenValueShow           // Chwytak 2 | wartość kalibracji otwartego chwytaka
    lrDispencersCatch3ClosedValueShow                	:LREAL;         //  P030_Recipes.stActRecipe.stUBL.lrDispencersCatch3ClosedValueShow         // Chwytak 3 | wartość kalibracji zamkniętego chwytaka
    lrDispencersCatch3OpenValueShow                     :LREAL;         //  P030_Recipes.stActRecipe.stUBL.lrDispencersCatch3OpenValueShow           // Chwytak 3 | wartość kalibracji otwartego chwytaka
    lrDispencersCatch4ClosedValueShow                   :LREAL;         //  P030_Recipes.stActRecipe.stUBL.lrDispencersCatch4ClosedValueShow         // Chwytak 4 | wartość kalibracji zamkniętego chwytaka
    lrDispencersCatch4OpenValueShow                     :LREAL;         //  P030_Recipes.stActRecipe.stUBL.lrDispencersCatch4OpenValueShow          // Chwytak 4 | wartość kalibracji otwartego chwytaka
    lrDispencersCatchToleranceShow                      :LREAL;         //  P030_Recipes.stActRecipe.stUBL.lrDispencersCatchToleranceShow            // Tolerancja chwytaka [0-100%]      
                                              		                    //
	//Zbiorniki                                                         //
	bTank1MixerEnableShow								:BOOL;	   		//	P030_Recipes.stActRecipe.stUBL.bTank1MixerEnableShow				// Mieszadło
	bTankHeatingEnableShow								:BOOL;   		//	P030_Recipes.stActRecipe.stUBL.bTankHeatingEnableShow				// Grzanie                                     		
	iTankHeatingTempSVShow								:INT;			//	P030_Recipes.stActRecipe.stUBL.iTankHeatingTempSVShow				// Temperatura
	bTank1PressureEnableShow							:BOOL;  		//	P030_Recipes.stActRecipe.stUBL.bTank1PressureEnableShow			// Ciśnienie                                   		
	bTank1SupplyPumpEnableShow							:BOOL;  		//	P030_Recipes.stActRecipe.stUBL.bTank1SupplyPumpEnableShow			// Aktywacja pompy 1
	bTank2SupplyPumpEnableShow							:BOOL;  		//	P030_Recipes.stActRecipe.stUBL.bTank2SupplyPumpEnableShow			// Aktywacja pompy 2
	uTank1LevelSetpointShow								:UINT;			//	P030_Recipes.stActRecipe.stUBL.uTank1LevelSetpointShow				// [H] Wartość zadana masy do czujnika poziomu w zbiorniku nr 1
	uTank2LevelSetpointShow								:UINT;			//	P030_Recipes.stActRecipe.stUBL.uTank2LevelSetpointShow				// [H] Wartość zadana masy do czujnika poziomu w zbiorniku nr 2
	bTank1LevelSignalInvertShow							:BOOL;			//	P030_Recipes.stActRecipe.stUBL.bTank1LevelSignalInvertShow			// [H] Odwróć sygnał z czujnika zbiornika pierwszego
	bTank2LevelSignalInvertShow							:BOOL;			//	P030_Recipes.stActRecipe.stUBL.bTank2LevelSignalInvertShow			// [H] Odwróć sygnał z czujnika zbionirka drugiego
 	//Zbiorniki-dodatkowe
	bTankRainbowModeShow								:BOOL;			// Tryb 4 zbiorników                 

                          			                //
	//Waga                                           					//	
	bWeight1EnableShow									:BOOL;			//	P030_Recipes.stActRecipe.stUBL.bWeight1EnableShow					// Aktywacja
	lrWeightMassSVShow 									:LREAL;			//	P030_Recipes.stActRecipe.stUBL.lrWeightMassSVShow 					// Waga zadana 
	iWeight1ActuatorUpDelayShow							: INT;			//	P030_Recipes.stActRecipe.stUBL.iWeight1ActuatorUpDelayShow		// Opóźnienie podnoszenia wagi 1
	iWeight2ActuatorUpDelayShow							: INT;			//	P030_Recipes.stActRecipe.stUBL.iWeight2ActuatorUpDelayShow		// Opóźnienie podnoszenia wagi 2
	iWeight3ActuatorUpDelayShow							: INT;			//	P030_Recipes.stActRecipe.stUBL.iWeight3ActuatorUpDelayShow		// Opóźnienie podnoszenia wagi 3
	iWeight4ActuatorUpDelayShow							: INT;			//	P030_Recipes.stActRecipe.stUBL.iWeight4ActuatorUpDelayShow		// Opóźnienie podnoszenia wagi 4
	iWeight5ActuatorUpDelayShow							: INT;			//	P030_Recipes.stActRecipe.stUBL.iWeight5ActuatorUpDelayShow		// Opóźnienie podnoszenia wagi 5 
	iWeight6ActuatorUpDelayShow							: INT;			//	P030_Recipes.stActRecipe.stUBL.iWeight6ActuatorUpDelayShow		// Opóźnienie podnoszenia wagi 6
	                                                                    //
	//Korekcja wagi                                     			    //
	lrFormWeightShow 									:LREAL;			//	P030_Recipes.stActRecipe.stUBL.lrFormWeightShow 								// [H] Waga formatki
	lrMass1DensityShow									:LREAL;			//	P030_Recipes.stActRecipe.stUBL.lrMass1DensityShow								// [H] Gęstoć masy pierwszej fazy [g/ml]
	lrMass2DensityShow									:LREAL;			//	P030_Recipes.stActRecipe.stUBL.lrMass2DensityShow								// [H] Gęstoć masy drugiej fazy [g/ml]
	lrCupWeightShow										:LREAL;			//	P030_Recipes.stActRecipe.stUBL.lrCupWeightShow									// Waga opakowania (z platynką, zależnie od opakowania) [g]
	lrWholePackageWeightShow							:LREAL;			//	P030_Recipes.stActRecipe.stUBL.lrWholePackageWeightShow						// [H] Waga całego opakowania bez masy (kubeczek,platynka,nakrętka) [g]
	lrWeight1MeasurmentCorrectionShow					:LREAL;			//	P030_Recipes.stActRecipe.stUBL.lrWeight1MeasurmentCorrectionShow				// [H] Korekta wagi zmierzonej [g] , różnica pomiedzy wskazaniami wagi zewnętrznej a linią
	bDispencer1WeightCorrectionEnableShow				:BOOL;			//	P030_Recipes.stActRecipe.stUBL.bDispencer1WeightCorrectionEnableShow			// Aktywacja korekcji 1
	bDispencer2WeightCorrectionEnableShow				:BOOL;			//	P030_Recipes.stActRecipe.stUBL.bDispencer2WeightCorrectionEnableShow			// Aktywacja korekcji 2
	bDispencer3WeightCorrectionEnableShow				:BOOL;			//	P030_Recipes.stActRecipe.stUBL.bDispencer3WeightCorrectionEnableShow			// Aktywacja korekcji 3
	bDispencer4WeightCorrectionEnableShow				:BOOL;			//	P030_Recipes.stActRecipe.stUBL.bDispencer4WeightCorrectionEnableShow			// Aktywacja korekcji 4	
	lrWeightUpperToleranceShow							:LREAL;			//	P030_Recipes.stActRecipe.stUBL.lrWeightUpperToleranceShow						// Górny zakres wagi [g]
	lrWeightLowerToleranceShow							:LREAL;			//	P030_Recipes.stActRecipe.stUBL.lrWeightLowerToleranceShow						// Dolny zakres wagi [g]
    iWeightCorrectionNumberOfSamplesShow				:UINT:=2;		//	P030_Recipes.stActRecipe.stUBL.iWeightCorrectionNumberOfSamplesShow			// Ilość próbek korekcji [x] (1-20)

 	//Podajnik knotów                                               
	bWickFeederEnableShow								:BOOL;			//	P030_Recipes.stActRecipe.stUBL.bLidFeederEnableShow				// Zezwolenie na pracę podajnika platynek 
	lrWickFeederHeightPosSVShow							:LREAL;			//	P030_Recipes.stActRecipe.stUBL.lrLidFeederHeightPosSVShow			// Wysokość na której ma znajdować się podajnik platynek
	iWickFeederSorterTimeDelayOnShow					: INT;
	iWickFeederSorterTimeDelayOffShow					: INT;
	iWickFeederSorterTimeToEmptySleeveErrorShow			: INT;
                                                                       
	//Przeciąganie podajnika knotów                                   
	bWickFeederDragingStationEnableShow					:BOOL;			//	P030_Recipes.stActRecipe.stUBL.bLidFeederDragingStationEnableShow					// Aktywacja przeciagania formatek pod podajnikem płatynek
	lrWickFeederDragingStationVelocityShow				:LREAL; 		//	P030_Recipes.stActRecipe.stUBL.lrLidFeederDragingStationVelocityShow				// Prędkosć przeciągania formatek pod podajnikem płatynek [0-100 %]	
    lrWickFeederDragingStationAccelerationShow			:LREAL; 		//	P030_Recipes.stActRecipe.stUBL.lrLidFeederDragingStationAccelerationShow		// Przyspieszenie przeciągania formatek pod podajnikem płatynek 	
    lrWickFeederDragingStationDecelerationShow			:LREAL; 		//	P030_Recipes.stActRecipe.stUBL.lrLidFeederDragingStationDecelerationShow		// Zmniejszenie prędkości przeciągania formatek pod podajnikem płatynek 	
                                                                      
	//Podajnik platynek                                                 //
	bLidFeederEnableShow								:BOOL;			//	P030_Recipes.stActRecipe.stUBL.bLidFeederEnableShow				// Zezwolenie na pracę podajnika platynek 
	bLidFeederHeaterEnableShow							:BOOL;			//	P030_Recipes.stActRecipe.stUBL.bLidFeederHeaterEnableShow			// Zezwolenie na prace grzałki podajnika platynek 
	lrLidFeederHeightPosSVShow							:LREAL;			//	P030_Recipes.stActRecipe.stUBL.lrLidFeederHeightPosSVShow			// Wysokość na której ma znajdować się podajnik platynek
	iLidFeederHeatingTimeShow							:INT; 			//	P030_Recipes.stActRecipe.stUBL.iLidFeederHeatingTimeShow			// Czas zgrzewania wstępnego podajnika platynek [ms]
	iLidFeederTempHisteresisShow						:INT;			//	P030_Recipes.stActRecipe.stUBL.iLidFeederTempHisteresisShow		// Histereza poprawnej temperatury grzałki podajnika platynek 1 (+/- *C), po jej przekroczeniu grzałka wpada w błąd
	iLidFeeder1TempSVShow								:INT;			//	P030_Recipes.stActRecipe.stUBL.iLidFeeder1TempSVShow				// Temperatura zadana grzałki podajnika platynek 1
	iLidFeeder2TempSVShow								:INT;			//	P030_Recipes.stActRecipe.stUBL.iLidFeeder2TempSVShow				// Temperatura zadana grzałki podajnika platynek 2
                                                                        //
	//Przeciąganie podajnika platynek                                   //
	bLidFeederDragingStationEnableShow					: BOOL;			//	P030_Recipes.stActRecipe.stUBL.bLidFeederDragingStationEnableShow					// Aktywacja przeciagania formatek pod podajnikem płatynek
	lrLidFeederDragingStationVelocityShow				: LREAL; 		//	P030_Recipes.stActRecipe.stUBL.lrLidFeederDragingStationVelocityShow				// Prędkosć przeciągania formatek pod podajnikem płatynek [0-100 %]	
    lrLidFeederDragingStationAccelerationShow			: LREAL; 		//	P030_Recipes.stActRecipe.stUBL.lrLidFeederDragingStationAccelerationShow		// Przyspieszenie przeciągania formatek pod podajnikem płatynek 	
    lrLidFeederDragingStationDecelerationShow			: LREAL; 		//	P030_Recipes.stActRecipe.stUBL.lrLidFeederDragingStationDecelerationShow		// Zmniejszenie prędkości przeciągania formatek pod podajnikem płatynek 	

